C09042=1045.167,89.318,-85.987,170.316,36.397,156.850
C09043=1045.173,89.567,-86.006,170.318,36.398,156.851
C09044=1045.179,89.816,-86.025,170.319,36.400,156.851
C09045=1045.185,90.066,-86.044,170.321,36.401,156.851
C09046=1045.192,90.315,-86.063,170.324,36.403,156.851
C09047=1045.198,90.564,-86.081,170.325,36.404,156.852
C09048=1045.204,90.813,-86.101,170.327,36.406,156.852
C09049=1045.210,91.062,-86.119,170.329,36.407,156.852
C09050=1045.216,91.312,-86.138,170.330,36.408,156.853
C09051=1045.223,91.560,-86.158,170.332,36.410,156.853
C09052=1045.228,91.810,-86.177,170.334,36.411,156.853
C09053=1045.234,92.059,-86.196,170.336,36.413,156.853
C09054=1045.240,92.308,-86.215,170.338,36.415,156.854
C09055=1045.247,92.558,-86.235,170.340,36.416,156.854
C09056=1045.253,92.807,-86.254,170.341,36.417,156.854
C09057=1045.260,93.093,-86.275,170.343,36.419,156.855
C09058=1045.267,93.379,-86.297,170.346,36.421,156.855
C09059=1045.274,93.665,-86.319,170.348,36.422,156.855
C09060=1045.281,93.951,-86.341,170.350,36.424,156.855
C09061=1045.288,94.200,-86.361,170.352,36.425,156.856
C09062=1045.293,94.449,-86.380,170.353,36.426,156.856
C09063=1045.300,94.698,-86.399,170.355,36.428,156.856
C09064=1045.305,94.948,-86.418,170.357,36.430,156.857
C09065=1045.312,95.196,-86.437,170.359,36.431,156.857
C09066=1045.318,95.446,-86.456,170.361,36.433,156.857
C09067=1045.324,95.695,-86.475,170.363,36.434,156.857
C09068=1045.331,95.944,-86.495,170.365,36.435,156.858
C09069=1045.337,96.193,-86.514,170.366,36.437,156.858
C09070=1045.343,96.443,-86.533,170.368,36.438,156.858
C09071=1045.349,96.692,-86.553,170.371,36.440,156.858
C09072=1045.355,96.941,-86.572,170.372,36.441,156.859
C09073=1045.361,97.190,-86.591,170.374,36.443,156.859
C09074=1045.368,97.439,-86.611,170.376,36.444,156.859
C09075=1045.373,97.688,-86.630,170.377,36.445,156.860
C09076=1045.381,97.938,-86.649,170.379,36.447,156.860
C09077=1045.386,98.153,-86.666,170.381,36.448,156.860
C09078=1045.391,98.367,-86.683,170.383,36.450,156.860
C09079=1045.396,98.582,-86.699,170.384,36.451,156.861
C09080=1045.401,98.797,-86.715,170.386,36.452,156.861
C09081=1045.407,99.011,-86.732,170.387,36.453,156.861
C09082=1045.412,99.227,-86.749,170.389,36.454,156.861
C09083=1045.418,99.441,-86.765,170.390,36.455,156.861
C09084=1045.423,99.655,-86.782,170.392,36.456,156.862
C09085=1045.429,99.905,-86.802,170.394,36.458,156.862
C09086=1045.436,100.153,-86.821,170.396,36.460,156.862
C09087=1045.442,100.403,-86.841,170.398,36.461,156.863
C09088=1045.448,100.653,-86.860,170.399,36.462,156.863
C09089=1045.454,100.901,-86.879,170.401,36.464,156.863
C09090=1045.460,101.150,-86.899,170.403,36.465,156.863
C09091=1045.466,101.400,-86.918,170.405,36.467,156.864
C09092=1045.472,101.648,-86.938,170.407,36.468,156.864
C09093=1045.478,101.899,-86.958,170.409,36.470,156.864
C09094=1045.485,102.147,-86.977,170.411,36.471,156.865
C09095=1045.491,102.397,-86.997,170.412,36.473,156.865
C09096=1045.497,102.645,-87.016,170.415,36.474,156.865
C09097=1045.503,102.895,-87.036,170.417,36.476,156.865
C09098=1045.509,103.144,-87.056,170.418,36.477,156.866
C09099=1045.515,103.394,-87.075,170.420,36.479,156.866
C09100=1045.522,103.642,-87.095,170.422,36.480,156.866
C09101=1045.528,103.891,-87.115,170.423,36.482,156.867
C09102=1045.533,104.140,-87.134,170.426,36.483,156.867
C09103=1045.539,104.389,-87.154,170.428,36.484,156.867
C09104=1045.546,104.639,-87.173,170.429,36.486,156.867
C09105=1045.552,104.888,-87.193,170.431,36.488,156.868
C09106=1045.558,105.137,-87.213,170.433,36.489,156.868
C09107=1045.564,105.386,-87.232,170.434,36.491,156.868
C09108=1045.571,105.636,-87.252,170.437,36.492,156.868
C09109=1045.577,105.885,-87.272,170.439,36.494,156.869
C09110=1045.582,106.134,-87.292,170.441,36.495,156.869
C09111=1045.588,106.383,-87.311,170.442,36.496,156.869
C09112=1045.596,106.632,-87.331,170.444,36.498,156.870
C09113=1045.601,106.881,-87.350,170.446,36.499,156.870
C09114=1045.607,107.130,-87.370,170.448,36.501,156.870
C09115=1045.613,107.379,-87.390,170.450,36.503,156.871
C09116=1045.620,107.629,-87.410,170.452,36.504,156.871
C09117=1045.626,107.878,-87.430,170.453,36.506,156.871
C09118=1045.632,108.126,-87.449,170.455,36.507,156.871
C09119=1045.639,108.376,-87.470,170.457,36.508,156.872
C09120=1045.645,108.625,-87.489,170.460,36.510,156.872
C09121=1045.654,108.980,-87.517,170.462,36.512,156.872
C09122=1045.662,109.335,-87.546,170.464,36.514,156.873
C09123=1045.671,109.689,-87.574,170.467,36.516,156.873
C09124=1045.680,110.044,-87.602,170.469,36.518,156.874
C09125=1045.686,110.294,-87.622,170.472,36.519,156.874
C09126=1045.692,110.542,-87.642,170.474,36.521,156.874
C09127=1045.698,110.791,-87.662,170.476,36.522,156.874
C09128=1045.705,111.041,-87.682,170.477,36.524,156.875
C09129=1045.711,111.290,-87.702,170.479,36.526,156.875
C09130=1045.716,111.539,-87.721,170.482,36.527,156.875
C09131=1045.723,111.789,-87.741,170.483,36.529,156.876
C09132=1045.729,112.037,-87.761,170.485,36.530,156.876
C09133=1045.735,112.286,-87.781,170.487,36.532,156.876
C09134=1045.742,112.536,-87.802,170.488,36.533,156.876
C09135=1045.748,112.785,-87.822,170.490,36.534,156.877
C09136=1045.754,113.033,-87.842,170.493,36.536,156.877
C09137=1045.760,113.283,-87.862,170.495,36.537,156.877
C09138=1045.766,113.532,-87.882,170.496,36.539,156.878
C09139=1045.772,113.780,-87.902,170.498,36.540,156.878
C09140=1045.778,114.031,-87.921,170.500,36.542,156.878
C09141=1045.784,114.280,-87.942,170.501,36.544,156.878
C09142=1045.790,114.529,-87.962,170.504,36.545,156.879
C09143=1045.796,114.778,-87.982,170.506,36.547,156.879
C09144=1045.803,115.026,-88.003,170.508,36.548,156.879
C09145=1045.808,115.275,-88.024,170.509,36.550,156.880
C09146=1045.814,115.525,-88.044,170.511,36.552,156.880
C09147=1045.820,115.774,-88.064,170.514,36.553,156.880
C09148=1045.826,116.023,-88.084,170.515,36.555,156.881
C09149=1045.832,116.272,-88.105,170.517,36.556,156.881
C09150=1045.838,116.521,-88.125,170.519,36.558,156.881
C09151=1045.844,116.770,-88.145,170.520,36.559,156.881
C09152=1045.850,117.020,-88.166,170.522,36.561,156.882
C09153=1045.856,117.269,-88.185,170.525,36.562,156.882
C09154=1045.862,117.517,-88.205,170.527,36.564,156.882
C09155=1045.868,117.767,-88.226,170.528,36.566,156.883
C09156=1045.874,118.016,-88.246,170.530,36.567,156.883
C09157=1045.880,118.265,-88.266,170.532,36.569,156.883
C09158=1045.887,118.514,-88.287,170.535,36.570,156.884
C09159=1045.892,118.763,-88.308,170.536,36.572,156.884
C09160=1045.899,119.012,-88.328,170.538,36.573,156.884
C09161=1045.905,119.261,-88.348,170.540,36.575,156.885
C09162=1045.910,119.510,-88.369,170.541,36.576,156.885
C09163=1045.917,119.760,-88.389,170.544,36.578,156.885
C09164=1045.923,120.009,-88.409,170.546,36.579,156.885
C09165=1045.929,120.258,-88.430,170.548,36.581,156.886
C09166=1045.935,120.507,-88.451,170.549,36.583,156.886
C09167=1045.941,120.756,-88.471,170.551,36.584,156.886
C09168=1045.947,121.005,-88.491,170.553,36.586,156.887
C09169=1045.953,121.254,-88.511,170.556,36.588,156.887
C09170=1045.959,121.503,-88.532,170.557,36.589,156.887
C09171=1045.965,121.752,-88.552,170.559,36.591,156.888
C09172=1045.971,122.002,-88.573,170.561,36.592,156.888
C09173=1045.977,122.251,-88.593,170.562,36.594,156.888
C09174=1045.984,122.499,-88.614,170.564,36.595,156.888
C09175=1045.989,122.749,-88.635,170.567,36.597,156.889
C09176=1045.996,122.998,-88.655,170.569,36.598,156.889
C09177=1046.002,123.247,-88.675,170.570,36.600,156.889
C09178=1046.008,123.496,-88.697,170.572,36.601,156.890
C09179=1046.014,123.745,-88.717,170.574,36.603,156.890
C09180=1046.021,123.994,-88.737,170.577,36.604,156.890
C09181=1046.026,124.243,-88.758,170.579,36.606,156.891
C09182=1046.033,124.492,-88.779,170.580,36.607,156.891
C09183=1046.039,124.741,-88.799,170.582,36.609,156.891
C09184=1046.045,124.990,-88.820,170.584,36.610,156.891
C09185=1046.052,125.276,-88.843,170.587,36.612,156.892
C09186=1046.059,125.562,-88.867,170.589,36.614,156.892
C09187=1046.066,125.848,-88.891,170.591,36.616,156.893
C09188=1046.073,126.133,-88.915,170.593,36.617,156.893
C09189=1046.079,126.382,-88.935,170.595,36.619,156.893
C09190=1046.085,126.632,-88.955,170.597,36.620,156.893
C09191=1046.092,126.881,-88.976,170.599,36.622,156.894
C09192=1046.098,127.130,-88.996,170.601,36.623,156.894
C09193=1046.104,127.379,-89.018,170.603,36.625,156.894
C09194=1046.110,127.628,-89.038,170.605,36.626,156.895
C09195=1046.117,127.877,-89.058,170.606,36.628,156.895
C09196=1046.122,128.126,-89.080,170.609,36.630,156.895
C09197=1046.129,128.375,-89.100,170.611,36.631,156.896
C09198=1046.135,128.624,-89.122,170.613,36.633,156.896
C09199=1046.141,128.873,-89.142,170.615,36.634,156.896
C09200=1046.148,129.122,-89.163,170.616,36.636,156.896
C09201=1046.153,129.371,-89.183,170.619,36.637,156.897
C09202=1046.160,129.620,-89.204,170.621,36.639,156.897
C09203=1046.167,129.870,-89.225,170.623,36.640,156.897
C09204=1046.172,130.118,-89.246,170.624,36.642,156.898
C09205=1046.179,130.368,-89.266,170.626,36.643,156.898
C09206=1046.185,130.616,-89.287,170.629,36.645,156.898
C09207=1046.191,130.866,-89.308,170.631,36.646,156.898
C09208=1046.198,131.115,-89.329,170.633,36.648,156.899
C09209=1046.203,131.364,-89.349,170.634,36.649,156.899
C09210=1046.210,131.613,-89.370,170.636,36.651,156.899
C09211=1046.216,131.862,-89.391,170.638,36.652,156.900
C09212=1046.222,132.111,-89.413,170.641,36.654,156.900
C09213=1046.229,132.360,-89.434,170.643,36.656,156.900
C09214=1046.234,132.609,-89.454,170.644,36.657,156.901
C09215=1046.240,132.858,-89.476,170.646,36.659,156.901
C09216=1046.247,133.107,-89.497,170.648,36.660,156.901
C09217=1046.252,133.356,-89.517,170.651,36.662,156.902
C09218=1046.258,133.605,-89.539,170.653,36.664,156.902
C09219=1046.265,133.854,-89.560,170.654,36.665,156.902
C09220=1046.270,134.103,-89.581,170.656,36.667,156.903
C09221=1046.277,134.353,-89.602,170.658,36.668,156.903
C09222=1046.283,134.601,-89.623,170.661,36.670,156.903
C09223=1046.289,134.851,-89.644,170.663,36.672,156.904
C09224=1046.295,135.100,-89.665,170.664,36.673,156.904
C09225=1046.300,135.348,-89.687,170.666,36.675,156.904
C09226=1046.307,135.597,-89.708,170.668,36.676,156.904
C09227=1046.313,135.847,-89.729,170.671,36.678,156.905
C09228=1046.319,136.096,-89.750,170.673,36.680,156.905
C09229=1046.326,136.344,-89.771,170.674,36.681,156.905
C09230=1046.332,136.594,-89.793,170.676,36.683,156.906
C09231=1046.337,136.843,-89.813,170.678,36.684,156.906
C09232=1046.344,137.092,-89.834,170.681,36.686,156.906
C09233=1046.350,137.341,-89.856,170.683,36.688,156.907
C09234=1046.356,137.589,-89.877,170.684,36.689,156.907
C09235=1046.362,137.839,-89.899,170.686,36.691,156.907
C09236=1046.369,138.088,-89.920,170.688,36.693,156.908
C09237=1046.374,138.337,-89.940,170.691,36.694,156.908
C09238=1046.380,138.586,-89.962,170.693,36.696,156.908
C09239=1046.386,138.835,-89.984,170.695,36.697,156.909
C09240=1046.393,139.084,-90.005,170.696,36.699,156.909
C09241=1046.399,139.332,-90.026,170.698,36.701,156.909
C09242=1046.405,139.582,-90.048,170.701,36.702,156.910
C09243=1046.411,139.831,-90.069,170.703,36.704,156.910
C09244=1046.417,140.079,-90.090,170.705,36.706,156.910
C09245=1046.423,140.329,-90.111,170.706,36.707,156.911
C09246=1046.429,140.578,-90.133,170.708,36.709,156.911
C09247=1046.435,140.828,-90.155,170.711,36.711,156.911
C09248=1046.440,141.076,-90.176,170.713,36.712,156.912
C09249=1046.448,141.362,-90.201,170.715,36.714,156.912
C09250=1046.455,141.647,-90.225,170.717,36.716,156.912
C09251=1046.462,141.933,-90.250,170.720,36.718,156.913
C09252=1046.469,142.218,-90.275,170.722,36.720,156.913
C09253=1046.475,142.467,-90.296,170.724,36.721,156.913
C09254=1046.481,142.716,-90.318,170.726,36.723,156.914
C09255=1046.487,142.965,-90.339,170.728,36.725,156.914
C09256=1046.493,143.214,-90.361,170.731,36.727,156.914
C09257=1046.499,143.463,-90.382,170.733,36.728,156.915
C09258=1046.506,143.712,-90.404,170.734,36.730,156.915
C09259=1046.511,143.961,-90.425,170.736,36.732,156.915
C09260=1046.517,144.210,-90.447,170.738,36.733,156.916
C09261=1046.523,144.459,-90.469,170.741,36.735,156.916
C09262=1046.530,144.708,-90.490,170.743,36.737,156.916
C09263=1046.536,144.958,-90.512,170.745,36.738,156.917
C09264=1046.541,145.206,-90.533,170.746,36.740,156.917
C09265=1046.547,145.455,-90.555,170.748,36.741,156.917
C09266=1046.554,145.704,-90.577,170.751,36.743,156.918
C09267=1046.560,145.953,-90.599,170.753,36.745,156.918
C09268=1046.566,146.202,-90.620,170.755,36.746,156.918
C09269=1046.572,146.451,-90.642,170.757,36.748,156.919
C09270=1046.578,146.700,-90.663,170.759,36.749,156.919
C09271=1046.585,146.949,-90.684,170.762,36.751,156.919
C09272=1046.591,147.198,-90.706,170.763,36.753,156.920
C09273=1046.597,147.447,-90.729,170.765,36.754,156.920
C09274=1046.603,147.696,-90.751,170.767,36.756,156.920
C09275=1046.609,147.945,-90.772,170.770,36.758,156.921
C09276=1046.615,148.194,-90.793,170.772,36.760,156.921
C09277=1046.621,148.443,-90.816,170.774,36.761,156.921
C09278=1046.627,148.692,-90.837,170.776,36.763,156.922
C09279=1046.633,148.941,-90.859,170.777,36.765,156.922
C09280=1046.640,149.190,-90.881,170.780,36.767,156.922
C09281=1046.645,149.439,-90.904,170.782,36.768,156.923
C09282=1046.651,149.688,-90.925,170.784,36.770,156.923
C09283=1046.657,149.937,-90.947,170.786,36.771,156.923
C09284=1046.664,150.185,-90.969,170.788,36.773,156.924
C09285=1046.670,150.435,-90.991,170.791,36.775,156.924
C09286=1046.676,150.684,-91.012,170.793,36.776,156.924
C09287=1046.682,150.933,-91.035,170.795,36.778,156.925
C09288=1046.688,151.182,-91.057,170.796,36.780,156.925
C09289=1046.693,151.430,-91.078,170.799,36.782,156.925
C09290=1046.700,151.679,-91.100,170.801,36.784,156.926
C09291=1046.705,151.929,-91.123,170.803,36.785,156.926
C09292=1046.711,152.178,-91.144,170.805,36.787,156.926
C09293=1046.718,152.426,-91.167,170.807,36.789,156.927
C09294=1046.724,152.676,-91.188,170.810,36.790,156.927
C09295=1046.731,152.924,-91.211,170.812,36.792,156.928
C09296=1046.736,153.174,-91.233,170.814,36.793,156.928
C09297=1046.742,153.422,-91.255,170.815,36.795,156.928
C09298=1046.749,153.671,-91.277,170.818,36.797,156.929
C09299=1046.754,153.920,-91.298,170.820,36.799,156.929
C09300=1046.760,154.169,-91.321,170.822,36.801,156.929
C09301=1046.766,154.418,-91.343,170.824,36.802,156.930
C09302=1046.772,154.667,-91.365,170.826,36.804,156.930
C09303=1046.779,154.916,-91.387,170.829,36.806,156.930
C09304=1046.784,155.165,-91.410,170.831,36.808,156.931
C09305=1046.791,155.414,-91.431,170.833,36.809,156.931
C09306=1046.796,155.663,-91.454,170.835,36.811,156.931
C09307=1046.803,155.911,-91.477,170.838,36.813,156.932
C09308=1046.809,156.161,-91.498,170.839,36.814,156.932
C09309=1046.815,156.410,-91.521,170.841,36.816,156.932
C09310=1046.821,156.659,-91.543,170.843,36.818,156.933
C09311=1046.827,156.907,-91.565,170.845,36.820,156.933
C09312=1046.833,157.157,-91.587,170.848,36.822,156.933
C09313=1046.840,157.441,-91.613,170.850,36.823,156.934
C09314=1046.847,157.727,-91.638,170.853,36.825,156.934
C09315=1046.854,158.012,-91.664,170.855,36.828,156.935
C09316=1046.861,158.297,-91.689,170.858,36.829,156.935
C09317=1046.867,158.546,-91.712,170.860,36.831,156.935
C09318=1046.873,158.795,-91.734,170.862,36.833,156.936
C09319=1046.879,159.044,-91.756,170.864,36.835,156.936
C09320=1046.885,159.293,-91.779,170.867,36.837,156.937
C09321=1046.891,159.542,-91.801,170.869,36.838,156.937
C09322=1046.897,159.791,-91.824,170.871,36.840,156.937
C09323=1046.903,160.040,-91.846,170.873,36.842,156.938
C09324=1046.910,160.288,-91.869,170.876,36.843,156.938
C09325=1046.915,160.538,-91.891,170.878,36.845,156.938
C09326=1046.921,160.787,-91.914,170.879,36.847,156.939
C09327=1046.927,161.035,-91.936,170.881,36.849,156.939
C09328=1046.933,161.284,-91.959,170.883,36.851,156.939
C09329=1046.939,161.534,-91.981,170.886,36.853,156.940
C09330=1046.944,161.782,-92.004,170.888,36.854,156.940
C09331=1046.951,162.031,-92.027,170.890,36.856,156.941
C09332=1046.956,162.280,-92.049,170.893,36.859,156.941
C09333=1046.962,162.529,-92.072,170.895,36.861,156.941
C09334=1046.968,162.778,-92.095,170.897,36.862,156.942
C09335=1046.974,163.027,-92.118,170.899,36.864,156.942
C09336=1046.980,163.275,-92.141,170.901,36.866,156.942
C09337=1046.986,163.525,-92.163,170.904,36.868,156.943
C09338=1046.991,163.774,-92.186,170.906,36.870,156.943
C09339=1046.997,164.023,-92.209,170.908,36.872,156.944
C09340=1047.003,164.271,-92.232,170.910,36.873,156.944
C09341=1047.009,164.520,-92.254,170.913,36.875,156.944
C09342=1047.015,164.769,-92.277,170.914,36.877,156.945
C09343=1047.021,165.018,-92.300,170.916,36.879,156.945
C09344=1047.026,165.267,-92.323,170.918,36.881,156.946
C09345=1047.032,165.516,-92.346,170.921,36.883,156.946
C09346=1047.039,165.764,-92.368,170.923,36.885,156.946
C09347=1047.045,166.014,-92.392,170.925,36.887,156.947
C09348=1047.051,166.263,-92.414,170.927,36.889,156.947
C09349=1047.056,166.512,-92.437,170.930,36.890,156.947
C09350=1047.062,166.761,-92.460,170.932,36.892,156.948
C09351=1047.069,167.009,-92.483,170.934,36.894,156.948
C09352=1047.074,167.258,-92.506,170.936,36.896,156.949
C09353=1047.080,167.507,-92.529,170.939,36.898,156.949
C09354=1047.086,167.756,-92.552,170.941,36.899,156.949
C09355=1047.092,168.005,-92.574,170.943,36.902,156.950
C09356=1047.098,168.253,-92.597,170.945,36.904,156.950
C09357=1047.105,168.502,-92.621,170.948,36.906,156.951
C09358=1047.110,168.751,-92.644,170.950,36.907,156.951
C09359=1047.116,169.000,-92.667,170.952,36.909,156.951
C09360=1047.122,169.249,-92.690,170.954,36.911,156.952
C09361=1047.128,169.498,-92.713,170.957,36.913,156.952
C09362=1047.134,169.746,-92.735,170.959,36.915,156.952
C09363=1047.140,169.995,-92.758,170.961,36.916,156.953
C09364=1047.146,170.244,-92.782,170.963,36.918,156.953
C09365=1047.152,170.493,-92.805,170.966,36.921,156.954
C09366=1047.158,170.742,-92.828,170.968,36.923,156.954
C09367=1047.164,170.991,-92.851,170.970,36.924,156.954
C09368=1047.170,171.240,-92.873,170.972,36.926,156.955
C09369=1047.176,171.489,-92.896,170.975,36.928,156.955
C09370=1047.182,171.737,-92.920,170.977,36.930,156.956
C09371=1047.188,171.986,-92.943,170.979,36.932,156.956
C09372=1047.194,172.235,-92.966,170.981,36.933,156.956
C09373=1047.200,172.484,-92.989,170.984,36.935,156.957
C09374=1047.206,172.733,-93.013,170.986,36.937,156.957
C09375=1047.213,172.982,-93.035,170.988,36.940,156.957
C09376=1047.218,173.231,-93.058,170.991,36.941,156.958
C09377=1047.225,173.515,-93.086,170.994,36.943,156.958
C09378=1047.232,173.800,-93.111,170.996,36.946,156.959
C09379=1047.239,174.085,-93.138,170.999,36.947,156.959
C09380=1047.246,174.370,-93.165,171.002,36.950,156.960
C09381=1047.253,174.619,-93.188,171.004,36.952,156.960
C09382=1047.258,174.868,-93.211,171.006,36.953,156.960
C09383=1047.264,175.116,-93.234,171.008,36.955,156.961
C09384=1047.271,175.366,-93.258,171.011,36.957,156.961
C09385=1047.276,175.614,-93.281,171.013,36.959,156.962
C09386=1047.283,175.863,-93.304,171.015,36.961,156.962
C09387=1047.288,176.112,-93.327,171.018,36.963,156.962
C09388=1047.295,176.361,-93.351,171.020,36.965,156.963
C09389=1047.301,176.610,-93.374,171.023,36.967,156.963
C09390=1047.307,176.858,-93.396,171.025,36.969,156.963
C09391=1047.314,177.107,-93.421,171.028,36.970,156.964
C09392=1047.319,177.356,-93.443,171.030,36.972,156.964
C09393=1047.325,177.604,-93.467,171.032,36.975,156.965
C09394=1047.332,177.854,-93.490,171.034,36.976,156.965
C09395=1047.338,178.102,-93.514,171.037,36.978,156.965
C09396=1047.344,178.352,-93.537,171.039,36.980,156.966
C09397=1047.350,178.600,-93.561,171.041,36.982,156.966
C09398=1047.356,178.849,-93.584,171.043,36.984,156.967
C09399=1047.363,179.098,-93.608,171.046,36.985,156.967
C09400=1047.368,179.347,-93.631,171.049,36.988,156.967
C09401=1047.375,179.595,-93.654,171.051,36.990,156.968
C09402=1047.381,179.844,-93.677,171.053,36.991,156.968
C09403=1047.387,180.093,-93.701,171.056,36.993,156.969
C09404=1047.394,180.342,-93.724,171.058,36.995,156.969
C09405=1047.400,180.590,-93.748,171.060,36.997,156.969
C09406=1047.406,180.839,-93.771,171.062,36.999,156.970
C09407=1047.412,181.088,-93.795,171.065,37.001,156.970
C09408=1047.418,181.337,-93.819,171.068,37.003,156.971
C09409=1047.425,181.586,-93.842,171.070,37.005,156.971
C09410=1047.431,181.835,-93.866,171.073,37.007,156.971
C09411=1047.437,182.084,-93.889,171.075,37.008,156.972
C09412=1047.443,182.332,-93.913,171.077,37.011,156.972
C09413=1047.450,182.581,-93.937,171.079,37.013,156.973
C09414=1047.455,182.830,-93.960,171.082,37.014,156.973
C09415=1047.462,183.079,-93.984,171.085,37.016,156.973
C09416=1047.469,183.327,-94.007,171.087,37.018,156.974
C09417=1047.475,183.577,-94.030,171.089,37.020,156.974
C09418=1047.481,183.825,-94.054,171.092,37.022,156.975
C09419=1047.486,184.074,-94.078,171.094,37.024,156.975
C09420=1047.493,184.323,-94.102,171.096,37.026,156.975
C09421=1047.498,184.572,-94.125,171.099,37.028,156.976
C09422=1047.505,184.821,-94.149,171.102,37.030,156.976
C09423=1047.510,185.069,-94.174,171.104,37.032,156.977
C09424=1047.516,185.318,-94.197,171.106,37.034,156.977
C09425=1047.523,185.567,-94.221,171.109,37.037,156.978
C09426=1047.528,185.815,-94.246,171.111,37.038,156.978
C09427=1047.535,186.064,-94.270,171.113,37.041,156.978
C09428=1047.540,186.313,-94.293,171.116,37.043,156.979
C09429=1047.546,186.562,-94.317,171.118,37.045,156.979
C09430=1047.552,186.811,-94.342,171.121,37.047,156.980
C09431=1047.558,187.059,-94.365,171.123,37.049,156.980
C09432=1047.563,187.309,-94.390,171.126,37.051,156.981
C09433=1047.570,187.557,-94.413,171.128,37.054,156.981
C09434=1047.575,187.806,-94.438,171.130,37.055,156.982
C09435=1047.581,188.054,-94.462,171.133,37.058,156.982
C09436=1047.587,188.304,-94.486,171.135,37.060,156.982
C09437=1047.593,188.552,-94.510,171.138,37.062,156.983
C09438=1047.599,188.801,-94.534,171.141,37.064,156.983
C09439=1047.605,189.050,-94.558,171.143,37.066,156.984
C09440=1047.611,189.298,-94.583,171.145,37.068,156.984
C09441=1047.618,189.582,-94.611,171.148,37.070,156.985
C09442=1047.625,189.867,-94.638,171.151,37.073,156.985
C09443=1047.631,190.151,-94.665,171.154,37.075,156.986
C09444=1047.638,190.436,-94.694,171.156,37.078,156.986
C09445=1047.645,190.685,-94.718,171.159,37.080,156.987
C09446=1047.650,190.933,-94.742,171.161,37.082,156.987
C09447=1047.657,191.182,-94.766,171.164,37.084,156.988
C09448=1047.662,191.431,-94.790,171.167,37.086,156.988
C09449=1047.669,191.680,-94.814,171.169,37.088,156.988
C09450=1047.674,191.929,-94.839,171.171,37.090,156.989
C09451=1047.681,192.177,-94.863,171.174,37.093,156.989
C09452=1047.687,192.426,-94.888,171.177,37.094,156.990
C09453=1047.693,192.675,-94.912,171.179,37.097,156.990
C09454=1047.699,192.924,-94.936,171.182,37.099,156.991
C09455=1047.705,193.172,-94.960,171.184,37.101,156.991
C09456=1047.711,193.421,-94.985,171.186,37.103,156.992
C09457=1047.717,193.669,-95.009,171.189,37.105,156.992
C09458=1047.723,193.918,-95.033,171.192,37.108,156.992
C09459=1047.730,194.167,-95.057,171.194,37.109,156.993
C09460=1047.735,194.416,-95.082,171.196,37.112,156.993
C09461=1047.741,194.665,-95.107,171.200,37.114,156.994
C09462=1047.748,194.914,-95.131,171.202,37.116,156.994
C09463=1047.753,195.162,-95.155,171.204,37.118,156.995
C09464=1047.760,195.411,-95.179,171.207,37.120,156.995
C09465=1047.765,195.659,-95.204,171.209,37.123,156.996
C09466=1047.772,195.908,-95.228,171.212,37.124,156.996
C09467=1047.778,196.157,-95.253,171.215,37.127,156.996
C09468=1047.785,196.406,-95.278,171.217,37.129,156.997
C09469=1047.790,196.654,-95.302,171.219,37.131,156.997
C09470=1047.796,196.904,-95.327,171.222,37.133,156.998
C09471=1047.803,197.152,-95.351,171.225,37.135,156.998
C09472=1047.808,197.401,-95.376,171.227,37.138,156.999
C09473=1047.815,197.649,-95.400,171.230,37.140,156.999
C09474=1047.821,197.898,-95.425,171.233,37.142,157.000
C09475=1047.827,198.146,-95.449,171.235,37.144,157.000
C09476=1047.833,198.395,-95.474,171.237,37.146,157.001
C09477=1047.839,198.644,-95.499,171.241,37.148,157.001
C09478=1047.846,198.893,-95.523,171.243,37.151,157.002
C09479=1047.851,199.141,-95.548,171.245,37.153,157.002
C09480=1047.858,199.390,-95.572,171.249,37.155,157.002
C09481=1047.864,199.639,-95.597,171.251,37.157,157.003
C09482=1047.870,199.888,-95.622,171.253,37.159,157.003
C09483=1047.876,200.136,-95.646,171.256,37.162,157.004
C09484=1047.882,200.385,-95.671,171.259,37.163,157.004
C09485=1047.889,200.634,-95.695,171.261,37.166,157.005
C09486=1047.895,200.883,-95.720,171.264,37.168,157.005
C09487=1047.901,201.132,-95.745,171.267,37.170,157.006
C09488=1047.908,201.379,-95.770,171.269,37.172,157.006
C09489=1047.914,201.628,-95.794,171.272,37.175,157.007
C09490=1047.920,201.877,-95.820,171.275,37.177,157.007
C09491=1047.926,202.126,-95.844,171.277,37.179,157.008
C09492=1047.931,202.374,-95.869,171.279,37.181,157.008
C09493=1047.938,202.623,-95.895,171.282,37.184,157.009
C09494=1047.943,202.872,-95.919,171.285,37.186,157.009
C09495=1047.950,203.121,-95.945,171.288,37.188,157.010
C09496=1047.957,203.369,-95.969,171.290,37.191,157.010
C09497=1047.962,203.618,-95.994,171.293,37.193,157.010
C09498=1047.968,203.867,-96.019,171.296,37.195,157.011
C09499=1047.974,204.115,-96.044,171.298,37.197,157.011
C09500=1047.981,204.364,-96.070,171.301,37.200,157.012
C09501=1047.986,204.613,-96.094,171.304,37.202,157.012
C09502=1047.992,204.861,-96.119,171.306,37.205,157.013
C09503=1047.998,205.110,-96.144,171.309,37.207,157.013
C09504=1048.004,205.359,-96.170,171.312,37.209,157.014
C09505=1048.030,206.410,-96.276,171.553,37.308,157.036
C09506=1048.037,206.675,-96.304,171.556,37.311,157.037
C09507=1048.044,206.939,-96.331,171.558,37.314,157.038
C09508=1048.051,207.204,-96.359,171.560,37.317,157.038
C09509=1048.058,207.469,-96.387,171.562,37.321,157.039
C09510=1048.065,207.717,-96.413,171.565,37.324,157.040
C09511=1048.071,207.965,-96.439,171.566,37.327,157.040
C09512=1048.077,208.215,-96.466,171.569,37.330,157.041
C09513=1048.084,208.463,-96.492,171.570,37.333,157.042
C09514=1048.091,208.711,-96.518,171.573,37.336,157.042
C09515=1048.097,208.960,-96.544,171.574,37.339,157.043
C09516=1048.103,209.208,-96.571,171.576,37.342,157.044
C09517=1048.110,209.457,-96.597,171.579,37.345,157.044
C09518=1048.117,209.705,-96.623,171.580,37.348,157.045
C09519=1048.123,209.954,-96.650,171.583,37.352,157.046
C09520=1048.129,210.202,-96.676,171.584,37.355,157.046
C09521=1048.136,210.451,-96.703,171.587,37.358,157.047
C09522=1048.142,210.700,-96.729,171.588,37.361,157.048
C09523=1048.149,210.948,-96.755,171.591,37.364,157.048
C09524=1048.155,211.197,-96.782,171.593,37.367,157.049
C09525=1048.162,211.445,-96.808,171.595,37.370,157.050
C09526=1048.169,211.693,-96.834,171.597,37.373,157.050
C09527=1048.175,211.942,-96.861,171.599,37.376,157.051
C09528=1048.182,212.191,-96.887,171.601,37.379,157.052
C09529=1048.187,212.439,-96.914,171.604,37.382,157.052
C09530=1048.195,212.688,-96.941,171.605,37.386,157.053
C09531=1048.200,212.936,-96.967,171.608,37.389,157.054
C09532=1048.207,213.185,-96.994,171.609,37.392,157.054
C09533=1048.213,213.433,-97.020,171.612,37.395,157.055
C09534=1048.220,213.682,-97.047,171.614,37.398,157.055
C09535=1048.226,213.930,-97.073,171.616,37.401,157.056
C09536=1048.232,214.179,-97.100,171.618,37.404,157.057
C09537=1048.239,214.427,-97.126,171.619,37.407,157.058
C09538=1048.246,214.676,-97.154,171.622,37.410,157.058
C09539=1048.252,214.924,-97.180,171.624,37.413,157.059
C09540=1048.259,215.173,-97.207,171.626,37.416,157.059
C09541=1048.264,215.421,-97.234,171.628,37.420,157.060
C09542=1048.271,215.670,-97.260,171.631,37.423,157.061
C09543=1048.277,215.918,-97.287,171.632,37.426,157.061
C09544=1048.284,216.167,-97.313,171.635,37.429,157.062
C09545=1048.290,216.415,-97.341,171.637,37.432,157.063
C09546=1048.298,216.664,-97.367,171.639,37.435,157.063
C09547=1048.303,216.912,-97.394,171.641,37.438,157.064
C09548=1048.310,217.161,-97.421,171.643,37.441,157.065
C09549=1048.316,217.409,-97.447,171.645,37.444,157.065
C09550=1048.323,217.658,-97.475,171.648,37.447,157.066
C09551=1048.330,217.906,-97.501,171.649,37.450,157.067
C09552=1048.336,218.155,-97.528,171.652,37.453,157.067
C09553=1048.342,218.404,-97.555,171.654,37.456,157.068
C09554=1048.349,218.651,-97.581,171.656,37.459,157.069
C09555=1048.355,218.900,-97.608,171.658,37.462,157.069
C09556=1048.362,219.149,-97.635,171.661,37.465,157.070
C09557=1048.369,219.397,-97.662,171.663,37.468,157.071
C09558=1048.375,219.646,-97.689,171.665,37.471,157.071
C09559=1048.382,219.894,-97.716,171.667,37.474,157.072
C09560=1048.388,220.142,-97.743,171.670,37.477,157.073
C09561=1048.395,220.391,-97.769,171.671,37.480,157.073
C09562=1048.402,220.661,-97.799,171.673,37.483,157.074
C09563=1048.409,220.931,-97.828,171.676,37.487,157.075
C09564=1048.416,221.201,-97.857,171.679,37.490,157.075
C09565=1048.422,221.471,-97.887,171.681,37.493,157.076
C09566=1048.429,221.720,-97.914,171.683,37.496,157.077
C09567=1048.435,221.967,-97.941,171.685,37.499,157.077
C09568=1048.442,222.216,-97.968,171.688,37.503,157.078
C09569=1048.449,222.465,-97.996,171.689,37.506,157.079
C09570=1048.454,222.713,-98.022,171.692,37.509,157.079
C09571=1048.461,222.962,-98.050,171.694,37.512,157.080
C09572=1048.467,223.211,-98.077,171.697,37.515,157.081
C09573=1048.473,223.458,-98.104,171.698,37.518,157.081
C09574=1048.481,223.707,-98.131,171.700,37.521,157.082
C09575=1048.487,223.956,-98.159,171.703,37.524,157.083
C09576=1048.493,224.204,-98.185,171.705,37.527,157.083
C09577=1048.500,224.452,-98.213,171.707,37.530,157.084
C09578=1048.506,224.701,-98.241,171.709,37.533,157.085
C09579=1048.512,224.949,-98.267,171.712,37.536,157.085
C09580=1048.519,225.198,-98.295,171.713,37.539,157.086
C09581=1048.526,225.446,-98.322,171.716,37.542,157.087
C09582=1048.532,225.694,-98.349,171.718,37.545,157.087
C09583=1048.539,225.943,-98.377,171.721,37.548,157.088
C09584=1048.545,226.192,-98.404,171.722,37.552,157.089
C09585=1048.551,226.439,-98.431,171.725,37.554,157.089
C09586=1048.558,226.688,-98.459,171.727,37.557,157.090
C09587=1048.564,226.937,-98.486,171.730,37.560,157.091
C09588=1048.571,227.185,-98.513,171.732,37.563,157.091
C09589=1048.577,227.433,-98.541,171.734,37.566,157.092
C09590=1048.584,227.682,-98.567,171.736,37.569,157.093
C09591=1048.591,227.930,-98.595,171.739,37.572,157.093
C09592=1048.597,228.179,-98.623,171.741,37.575,157.094
C09593=1048.604,228.428,-98.650,171.743,37.578,157.095
C09594=1048.610,228.675,-98.677,171.745,37.581,157.095
C09595=1048.617,228.924,-98.705,171.748,37.584,157.096
C09596=1048.623,229.172,-98.733,171.750,37.587,157.097
C09597=1048.630,229.421,-98.760,171.753,37.590,157.097
C09598=1048.636,229.669,-98.787,171.754,37.593,157.098
C09599=1048.642,229.918,-98.815,171.757,37.596,157.099
C09600=1048.649,230.166,-98.842,171.759,37.599,157.099
C09601=1048.655,230.415,-98.871,171.762,37.602,157.100
C09602=1048.662,230.663,-98.898,171.764,37.605,157.101
C09603=1048.668,230.911,-98.926,171.766,37.608,157.101
C09604=1048.674,231.160,-98.953,171.768,37.611,157.102
C09605=1048.681,231.409,-98.981,171.771,37.614,157.102
C09606=1048.688,231.657,-99.008,171.773,37.618,157.103
C09607=1048.694,231.905,-99.036,171.776,37.621,157.104
C09608=1048.700,232.153,-99.063,171.777,37.624,157.105
C09609=1048.706,232.402,-99.092,171.780,37.627,157.105
C09610=1048.713,232.650,-99.119,171.782,37.629,157.106
C09611=1048.720,232.899,-99.147,171.785,37.632,157.107
C09612=1048.726,233.147,-99.175,171.787,37.635,157.107
C09613=1048.732,233.395,-99.203,171.790,37.638,157.108
C09614=1048.738,233.644,-99.231,171.791,37.641,157.108
C09615=1048.745,233.892,-99.258,171.794,37.645,157.109
C09616=1048.752,234.141,-99.286,171.796,37.648,157.110
C09617=1048.758,234.389,-99.314,171.799,37.651,157.111
C09618=1048.764,234.651,-99.344,171.801,37.654,157.111
C09619=1048.772,234.914,-99.373,171.804,37.657,157.112
C09620=1048.778,235.176,-99.403,171.806,37.660,157.113
C09621=1048.785,235.438,-99.432,171.809,37.663,157.113
C09622=1048.791,235.687,-99.459,171.811,37.667,157.114
C09623=1048.797,235.936,-99.488,171.814,37.670,157.115
C09624=1048.804,236.183,-99.516,171.815,37.673,157.115
C09625=1048.811,236.432,-99.544,171.818,37.675,157.116
C09626=1048.818,236.680,-99.572,171.820,37.678,157.117
C09627=1048.824,236.929,-99.600,171.823,37.681,157.117
C09628=1048.830,237.178,-99.628,171.825,37.684,157.118
C09629=1048.837,237.426,-99.655,171.828,37.687,157.119
C09630=1048.843,237.673,-99.684,171.830,37.690,157.119
C09631=1048.849,237.922,-99.712,171.833,37.693,157.120
C09632=1048.856,238.170,-99.740,171.834,37.696,157.121
C09633=1048.862,238.419,-99.768,171.837,37.700,157.121
C09634=1048.869,238.667,-99.796,171.840,37.702,157.122
C09635=1048.876,238.915,-99.824,171.842,37.705,157.123
C09636=1048.882,239.164,-99.852,171.845,37.708,157.123
C09637=1048.888,239.413,-99.880,171.847,37.711,157.124
C09638=1048.895,239.660,-99.909,171.850,37.714,157.125
C09639=1048.901,239.909,-99.937,171.852,37.717,157.125
C09640=1048.908,240.158,-99.965,171.855,37.720,157.126
C09641=1048.915,240.406,-99.992,171.857,37.723,157.127
C09642=1048.921,240.654,-100.021,171.860,37.726,157.127
C09643=1048.928,240.903,-100.049,171.862,37.729,157.128
C09644=1048.934,241.151,-100.078,171.864,37.732,157.129
C09645=1048.940,241.399,-100.106,171.866,37.735,157.129
C09646=1048.947,241.648,-100.134,171.869,37.738,157.130
C09647=1048.953,241.896,-100.163,171.871,37.741,157.131
C09648=1048.959,242.144,-100.191,171.874,37.744,157.131
C09649=1048.966,242.392,-100.219,171.876,37.747,157.132
C09650=1048.972,242.641,-100.248,171.879,37.750,157.133
C09651=1048.979,242.889,-100.276,171.881,37.753,157.133
C09652=1048.985,243.138,-100.305,171.884,37.756,157.134
C09653=1048.991,243.386,-100.334,171.886,37.759,157.135
C09654=1048.998,243.634,-100.361,171.889,37.762,157.135
C09655=1049.004,243.882,-100.390,171.891,37.765,157.136
C09656=1049.011,244.131,-100.418,171.894,37.768,157.137
C09657=1049.017,244.379,-100.447,171.896,37.771,157.137
C09658=1049.023,244.628,-100.475,171.899,37.774,157.138
C09659=1049.030,244.875,-100.504,171.901,37.777,157.139
C09660=1049.036,245.124,-100.533,171.904,37.780,157.139
C09661=1049.043,245.372,-100.561,171.906,37.783,157.140
C09662=1049.049,245.620,-100.590,171.909,37.786,157.141
C09663=1049.055,245.869,-100.618,171.911,37.789,157.141
C09664=1049.062,246.117,-100.647,171.914,37.792,157.142
C09665=1049.069,246.365,-100.676,171.916,37.795,157.143
C09666=1049.075,246.614,-100.704,171.918,37.799,157.143
C09667=1049.081,246.862,-100.733,171.921,37.802,157.144
C09668=1049.087,247.110,-100.762,171.923,37.804,157.145
C09669=1049.093,247.358,-100.791,171.926,37.807,157.145
C09670=1049.099,247.607,-100.819,171.928,37.811,157.146
C09671=1049.105,247.855,-100.848,171.931,37.814,157.147
C09672=1049.112,248.103,-100.877,171.933,37.817,157.148
C09673=1049.119,248.352,-100.906,171.936,37.820,157.148
C09674=1049.125,248.608,-100.936,171.938,37.823,157.149
C09675=1049.132,248.865,-100.965,171.941,37.826,157.150
C09676=1049.138,249.121,-100.996,171.944,37.829,157.150
C09677=1049.145,249.378,-101.025,171.947,37.833,157.151
C09678=1049.151,249.626,-101.055,171.950,37.835,157.152
C09679=1049.158,249.875,-101.084,171.952,37.838,157.152
C09680=1049.164,250.123,-101.113,171.955,37.841,157.153
C09681=1049.171,250.370,-101.141,171.957,37.844,157.154
C09682=1049.177,250.619,-101.170,171.960,37.848,157.155
C09683=1049.183,250.867,-101.198,171.962,37.851,157.155
C09684=1049.189,251.115,-101.227,171.965,37.854,157.156
C09685=1049.196,251.364,-101.257,171.967,37.856,157.157
C09686=1049.202,251.612,-101.286,171.970,37.859,157.157
C09687=1049.209,251.861,-101.315,171.972,37.863,157.158
C09688=1049.215,252.109,-101.344,171.975,37.866,157.159
C09689=1049.221,252.357,-101.373,171.977,37.869,157.159
C09690=1049.228,252.605,-101.401,171.980,37.872,157.160
C09691=1049.235,252.853,-101.431,171.982,37.875,157.161
C09692=1049.241,253.102,-101.460,171.985,37.877,157.161
C09693=1049.248,253.350,-101.489,171.988,37.881,157.162
C09694=1049.254,253.598,-101.518,171.990,37.884,157.163
C09695=1049.260,253.846,-101.547,171.993,37.887,157.163
C09696=1049.267,254.095,-101.576,171.996,37.890,157.164
C09697=1049.273,254.343,-101.605,171.999,37.893,157.165
C09698=1049.279,254.591,-101.635,172.001,37.895,157.165
C09699=1049.286,254.839,-101.664,172.004,37.899,157.166
C09700=1049.293,255.087,-101.694,172.006,37.902,157.167
C09701=1049.299,255.336,-101.723,172.009,37.905,157.167
C09702=1049.306,255.583,-101.751,172.011,37.908,157.168
C09703=1049.312,255.832,-101.780,172.014,37.911,157.169
C09704=1049.319,256.080,-101.810,172.016,37.914,157.169
C09705=1049.325,256.329,-101.839,172.020,37.916,157.170
C09706=1049.332,256.577,-101.868,172.023,37.920,157.171
C09707=1049.339,256.825,-101.898,172.025,37.923,157.172
C09708=1049.345,257.073,-101.927,172.028,37.926,157.172
C09709=1049.351,257.321,-101.956,172.030,37.929,157.173
C09710=1049.358,257.569,-101.985,172.033,37.932,157.174
C09711=1049.365,257.817,-102.015,172.035,37.934,157.174
C09712=1049.371,258.066,-102.044,172.038,37.937,157.175
C09713=1049.377,258.314,-102.073,172.041,37.940,157.176
C09714=1049.384,258.563,-102.103,172.044,37.944,157.176
C09715=1049.391,258.810,-102.132,172.046,37.947,157.177
C09716=1049.397,259.059,-102.162,172.049,37.950,157.178
C09717=1049.404,259.307,-102.191,172.052,37.952,157.178
C09718=1049.410,259.555,-102.221,172.054,37.955,157.179
C09719=1049.417,259.803,-102.250,172.058,37.958,157.180
C09720=1049.423,260.052,-102.279,172.060,37.961,157.180
C09721=1049.430,260.299,-102.309,172.063,37.964,157.181
C09722=1049.437,260.548,-102.338,172.065,37.967,157.182
C09723=1049.444,260.796,-102.367,172.068,37.970,157.182
C09724=1049.451,261.044,-102.397,172.070,37.973,157.183
C09725=1049.457,261.292,-102.426,172.074,37.976,157.184
C09726=1049.464,261.540,-102.456,172.076,37.979,157.184
C09727=1049.471,261.788,-102.485,172.079,37.982,157.185
C09728=1049.477,262.036,-102.514,172.081,37.985,157.186
C09729=1049.484,262.285,-102.544,172.085,37.988,157.186
C09730=1049.491,262.540,-102.575,172.088,37.991,157.187
C09731=1049.497,262.794,-102.605,172.090,37.994,157.188
C09732=1049.504,263.050,-102.635,172.093,37.997,157.189
C09733=1049.511,263.305,-102.666,172.096,38.000,157.189
C09734=1049.516,263.553,-102.696,172.099,38.003,157.190
C09735=1049.523,263.801,-102.726,172.101,38.006,157.191
C09736=1049.530,264.049,-102.755,172.104,38.010,157.192
C09737=1049.536,264.297,-102.786,172.107,38.013,157.192
C09738=1049.542,264.546,-102.815,172.110,38.015,157.193
C09739=1049.549,264.794,-102.845,172.113,38.018,157.194
C09740=1049.555,265.042,-102.876,172.115,38.022,157.194
C09741=1049.562,265.290,-102.905,172.118,38.025,157.195
C09742=1049.568,265.538,-102.934,172.120,38.028,157.196
C09743=1049.575,265.786,-102.965,172.124,38.030,157.196
C09744=1049.581,266.034,-102.995,172.127,38.034,157.197
C09745=1049.588,266.283,-103.024,172.129,38.037,157.198
C09746=1049.594,266.530,-103.055,172.132,38.040,157.198
C09747=1049.601,266.779,-103.085,172.135,38.043,157.199
C09748=1049.608,267.026,-103.115,172.138,38.046,157.200
C09749=1049.614,267.275,-103.145,172.140,38.049,157.201
C09750=1049.620,267.523,-103.174,172.143,38.052,157.201
C09751=1049.627,267.771,-103.204,172.147,38.055,157.202
C09752=1049.633,268.019,-103.235,172.149,38.058,157.203
C09753=1049.640,268.267,-103.265,172.152,38.061,157.203
C09754=1049.646,268.515,-103.295,172.154,38.064,157.204
C09755=1049.653,268.764,-103.325,172.158,38.067,157.205
C09756=1049.659,269.012,-103.355,172.160,38.070,157.206
C09757=1049.666,269.260,-103.385,172.163,38.073,157.206
C09758=1049.672,269.508,-103.415,172.166,38.077,157.207
C09759=1049.679,269.756,-103.446,172.169,38.080,157.208
C09760=1049.685,270.004,-103.476,172.172,38.082,157.208
C09761=1049.692,270.252,-103.506,172.174,38.086,157.209
C09762=1049.698,270.500,-103.537,172.178,38.089,157.210
C09763=1049.705,270.748,-103.567,172.180,38.092,157.211
C09764=1049.711,270.996,-103.597,172.183,38.095,157.211
C09765=1049.718,271.244,-103.627,172.186,38.098,157.212
C09766=1049.724,271.492,-103.658,172.189,38.101,157.213
C09767=1049.731,271.740,-103.687,172.192,38.104,157.213
C09768=1049.737,271.988,-103.718,172.194,38.107,157.214
C09769=1049.744,272.237,-103.749,172.198,38.110,157.215
C09770=1049.750,272.484,-103.779,172.201,38.113,157.216
C09771=1049.757,272.733,-103.809,172.203,38.116,157.216
C09772=1049.763,272.980,-103.840,172.207,38.120,157.217
C09773=1049.770,273.228,-103.871,172.209,38.123,157.218
C09774=1049.776,273.477,-103.901,172.212,38.126,157.218
C09775=1049.782,273.725,-103.932,172.216,38.129,157.219
C09776=1049.789,273.973,-103.962,172.218,38.132,157.220
C09777=1049.795,274.221,-103.992,172.221,38.135,157.221
C09778=1049.802,274.469,-104.024,172.224,38.138,157.221
C09779=1049.809,274.717,-104.054,172.227,38.141,157.222
C09780=1049.815,274.965,-104.084,172.229,38.145,157.223
C09781=1049.821,275.213,-104.115,172.233,38.147,157.224
C09782=1049.829,275.461,-104.146,172.236,38.150,157.224
C09783=1049.835,275.709,-104.176,172.238,38.154,157.225
C09784=1049.841,275.957,-104.207,172.242,38.157,157.226
C09785=1049.848,276.205,-104.238,172.244,38.160,157.227
C09786=1049.854,276.464,-104.270,172.248,38.163,157.227
C09787=1049.861,276.724,-104.302,172.251,38.166,157.228
C09788=1049.868,276.983,-104.334,172.253,38.170,157.229
C09789=1049.874,277.242,-104.366,172.257,38.173,157.229
C09790=1049.881,277.490,-104.396,172.260,38.176,157.230
C09791=1049.888,277.738,-104.428,172.263,38.179,157.231
C09792=1049.894,277.986,-104.458,172.266,38.182,157.232
C09793=1049.901,278.234,-104.489,172.268,38.185,157.232
C09794=1049.908,278.482,-104.520,172.272,38.189,157.233
C09795=1049.914,278.731,-104.550,172.275,38.192,157.234
C09796=1049.920,278.978,-104.581,172.278,38.194,157.235
C09797=1049.927,279.226,-104.612,172.281,38.198,157.235
C09798=1049.934,279.474,-104.644,172.283,38.201,157.236
C09799=1049.940,279.723,-104.674,172.287,38.204,157.237
C09800=1049.946,279.970,-104.705,172.290,38.207,157.238
C09801=1049.953,280.218,-104.737,172.293,38.210,157.238
C09802=1049.959,280.467,-104.767,172.296,38.213,157.239
C09803=1049.966,280.714,-104.799,172.298,38.217,157.240
C09804=1049.972,280.962,-104.829,172.302,38.220,157.241
C09805=1049.979,281.210,-104.861,172.305,38.223,157.241
C09806=1049.985,281.458,-104.892,172.308,38.226,157.242
C09807=1049.992,281.707,-104.923,172.311,38.229,157.243
C09808=1049.998,281.954,-104.954,172.315,38.233,157.244
C09809=1050.005,282.202,-104.985,172.317,38.236,157.244
C09810=1050.011,282.450,-105.016,172.320,38.239,157.245
C09811=1050.018,282.698,-105.047,172.323,38.242,157.246
C09812=1050.024,282.946,-105.079,172.326,38.245,157.247
C09813=1050.031,283.193,-105.110,172.330,38.248,157.247
C09814=1050.037,283.442,-105.141,172.332,38.252,157.248
C09815=1050.044,283.690,-105.172,172.336,38.255,157.249
C09816=1050.050,283.938,-105.204,172.339,38.258,157.250
C09817=1050.057,284.185,-105.235,172.342,38.261,157.250
C09818=1050.064,284.433,-105.266,172.345,38.264,157.251
C09819=1050.070,284.681,-105.297,172.349,38.267,157.252
C09820=1050.076,284.929,-105.328,172.351,38.270,157.253
C09821=1050.083,285.177,-105.360,172.355,38.274,157.253
C09822=1050.090,285.425,-105.391,172.357,38.277,157.254
C09823=1050.097,285.673,-105.422,172.361,38.280,157.255
C09824=1050.103,285.921,-105.454,172.364,38.283,157.256
C09825=1050.110,286.169,-105.485,172.367,38.286,157.256
C09826=1050.117,286.416,-105.517,172.370,38.290,157.257
C09827=1050.123,286.664,-105.548,172.374,38.293,157.258
C09828=1050.129,286.913,-105.580,172.376,38.296,157.259
C09829=1050.136,287.161,-105.611,172.380,38.299,157.260
C09830=1050.142,287.408,-105.642,172.382,38.302,157.260
C09831=1050.149,287.656,-105.673,172.386,38.306,157.261
C09832=1050.155,287.904,-105.705,172.389,38.308,157.262
C09833=1050.162,288.151,-105.737,172.392,38.312,157.263
C09834=1050.169,288.399,-105.768,172.395,38.315,157.263
C09835=1050.175,288.648,-105.800,172.399,38.318,157.264
C09836=1050.182,288.895,-105.832,172.401,38.322,157.265
C09837=1050.189,289.143,-105.863,172.405,38.325,157.266
C09838=1050.195,289.392,-105.895,172.408,38.328,157.266
C09839=1050.201,289.639,-105.927,172.411,38.331,157.267
C09840=1050.208,289.887,-105.958,172.414,38.335,157.268
C09841=1050.215,290.135,-105.990,172.418,38.337,157.269
C09842=1050.222,290.406,-106.025,172.421,38.341,157.270
C09843=1050.229,290.676,-106.060,172.424,38.345,157.270
C09844=1050.236,290.947,-106.094,172.428,38.348,157.271
C09845=1050.243,291.218,-106.129,172.431,38.352,157.272
C09846=1050.250,291.466,-106.161,172.435,38.355,157.273
C09847=1050.257,291.713,-106.193,172.438,38.358,157.274
C09848=1050.263,291.962,-106.225,172.442,38.362,157.275
C09849=1050.270,292.210,-106.256,172.444,38.365,157.275
C09850=1050.277,292.457,-106.288,172.448,38.368,157.276
C09851=1050.283,292.705,-106.320,172.451,38.371,157.277
C09852=1050.289,292.953,-106.352,172.454,38.375,157.278
C09853=1050.296,293.201,-106.385,172.458,38.378,157.278
C09854=1050.302,293.448,-106.416,172.460,38.381,157.279
C09855=1050.309,293.696,-106.447,172.464,38.385,157.280
C09856=1050.315,293.944,-106.480,172.468,38.388,157.281
C09857=1050.322,294.192,-106.512,172.470,38.391,157.282
C09858=1050.328,294.439,-106.544,172.474,38.394,157.282
C09859=1050.336,294.688,-106.576,172.477,38.398,157.283
C09860=1050.343,294.935,-106.608,172.481,38.401,157.284
C09861=1050.349,295.184,-106.640,172.484,38.404,157.285
C09862=1050.356,295.431,-106.673,172.487,38.408,157.286
C09863=1050.362,295.679,-106.705,172.490,38.411,157.286
C09864=1050.369,295.926,-106.737,172.493,38.414,157.287
C09865=1050.375,296.175,-106.769,172.497,38.417,157.288
C09866=1050.381,296.422,-106.801,172.501,38.421,157.289
C09867=1050.388,296.669,-106.834,172.503,38.424,157.290
C09868=1050.394,296.918,-106.866,172.507,38.428,157.290
C09869=1050.401,297.166,-106.899,172.511,38.431,157.291
C09870=1050.407,297.414,-106.932,172.513,38.434,157.292
C09871=1050.413,297.662,-106.964,172.517,38.438,157.293
C09872=1050.420,297.909,-106.996,172.520,38.441,157.294
C09873=1050.427,298.157,-107.028,172.524,38.445,157.295
C09874=1050.433,298.404,-107.061,172.527,38.448,157.295
C09875=1050.439,298.652,-107.094,172.530,38.451,157.296
C09876=1050.445,298.900,-107.126,172.534,38.455,157.297
C09877=1050.452,299.147,-107.158,172.537,38.458,157.298
C09878=1050.459,299.396,-107.191,172.540,38.461,157.299
C09879=1050.465,299.643,-107.224,172.544,38.465,157.299
C09880=1050.472,299.891,-107.257,172.547,38.468,157.300
C09881=1050.478,300.139,-107.289,172.550,38.472,157.301
C09882=1050.485,300.386,-107.321,172.554,38.475,157.302
C09883=1050.491,300.634,-107.354,172.558,38.478,157.303
C09884=1050.498,300.882,-107.387,172.560,38.482,157.304
C09885=1050.504,301.130,-107.419,172.564,38.485,157.304
C09886=1050.510,301.377,-107.452,172.568,38.489,157.305
C09887=1050.517,301.625,-107.484,172.571,38.493,157.306
C09888=1050.524,301.873,-107.517,172.574,38.496,157.307
C09889=1050.531,302.121,-107.550,172.578,38.499,157.308
C09890=1050.537,302.368,-107.583,172.582,38.503,157.309
C09891=1050.543,302.616,-107.616,172.584,38.506,157.310
C09892=1050.550,302.864,-107.649,172.588,38.509,157.310
C09893=1050.557,303.111,-107.681,172.592,38.513,157.311
C09894=1050.563,303.359,-107.714,172.595,38.516,157.312
C09895=1050.570,303.606,-107.746,172.598,38.520,157.313
C09896=1050.577,303.855,-107.780,172.602,38.523,157.314
C09897=1050.583,304.102,-107.812,172.606,38.526,157.315
C09898=1050.591,304.389,-107.850,172.610,38.530,157.315
C09899=1050.598,304.675,-107.889,172.613,38.534,157.316
C09900=1050.606,304.962,-107.926,172.617,38.539,157.318
C09901=1050.614,305.249,-107.965,172.621,38.543,157.319
C09902=1050.620,305.497,-107.998,172.625,38.546,157.319
C09903=1050.627,305.745,-108.031,172.629,38.549,157.320
C09904=1050.635,305.992,-108.064,172.632,38.553,157.321
C09905=1050.641,306.240,-108.096,172.636,38.556,157.322
C09906=1050.648,306.488,-108.129,172.639,38.559,157.323
C09907=1050.654,306.735,-108.162,172.642,38.563,157.324
C09908=1050.661,306.983,-108.196,172.646,38.567,157.324
C09909=1050.668,307.231,-108.229,172.650,38.570,157.325
C09910=1050.674,307.478,-108.262,172.654,38.573,157.326
C09911=1050.681,307.726,-108.295,172.656,38.577,157.327
C09912=1050.687,307.974,-108.328,172.660,38.580,157.328
C09913=1050.695,308.222,-108.361,172.664,38.584,157.329
C09914=1050.702,308.468,-108.394,172.668,38.587,157.330
C09915=1050.708,308.717,-108.427,172.671,38.591,157.330
C09916=1050.715,308.964,-108.461,172.674,38.594,157.331
C09917=1050.722,309.212,-108.494,172.678,38.598,157.332
C09918=1050.728,309.460,-108.526,172.682,38.601,157.333
C09919=1050.735,309.707,-108.560,172.686,38.605,157.334
C09920=1050.742,309.955,-108.593,172.689,38.608,157.335
C09921=1050.749,310.203,-108.627,172.693,38.611,157.336
C09922=1050.755,310.450,-108.660,172.697,38.615,157.336
C09923=1050.762,310.698,-108.693,172.700,38.619,157.337
C09924=1050.769,310.945,-108.726,172.703,38.622,157.338
C09925=1050.777,311.193,-108.759,172.707,38.625,157.339
C09926=1050.784,311.441,-108.793,172.711,38.629,157.340
C09927=1050.790,311.688,-108.826,172.714,38.632,157.341
C09928=1050.797,311.936,-108.860,172.718,38.636,157.342
C09929=1050.804,312.183,-108.893,172.722,38.639,157.343
C09930=1050.811,312.431,-108.926,172.726,38.643,157.343
C09931=1050.818,312.679,-108.959,172.730,38.647,157.344
C09932=1050.824,312.926,-108.993,172.732,38.650,157.345
C09933=1050.832,313.174,-109.027,172.736,38.653,157.346
C09934=1050.838,313.422,-109.061,172.740,38.657,157.347
C09935=1050.844,313.670,-109.094,172.744,38.661,157.348
C09936=1050.851,313.918,-109.128,172.748,38.665,157.349
C09937=1050.857,314.164,-109.162,172.751,38.668,157.350
C09938=1050.864,314.412,-109.196,172.755,38.672,157.351
C09939=1050.870,314.659,-109.230,172.759,38.676,157.352
C09940=1050.877,314.907,-109.264,172.762,38.679,157.352
C09941=1050.883,315.154,-109.298,172.766,38.683,157.353
C09942=1050.890,315.402,-109.332,172.769,38.686,157.354
C09943=1050.897,315.650,-109.366,172.773,38.690,157.355
C09944=1050.903,315.898,-109.399,172.777,38.694,157.356
C09945=1050.910,316.146,-109.433,172.781,38.698,157.357
C09946=1050.916,316.394,-109.467,172.785,38.701,157.358
C09947=1050.923,316.641,-109.501,172.788,38.705,157.359
C09948=1050.929,316.889,-109.535,172.792,38.709,157.360
C09949=1050.936,317.135,-109.569,172.796,38.713,157.361
C09950=1050.943,317.383,-109.604,172.799,38.716,157.362
C09951=1050.950,317.631,-109.638,172.803,38.720,157.363
C09952=1050.956,317.879,-109.672,172.807,38.724,157.364
C09953=1050.963,318.126,-109.706,172.810,38.727,157.364
C09954=1050.971,318.417,-109.746,172.815,38.732,157.366
C09955=1050.979,318.708,-109.786,172.819,38.736,157.367
C09956=1050.987,318.999,-109.826,172.824,38.740,157.368
C09957=1050.995,319.290,-109.866,172.828,38.745,157.369
C09958=1051.001,319.538,-109.901,172.832,38.748,157.370
C09959=1051.008,319.785,-109.934,172.836,38.752,157.371
C09960=1051.014,320.033,-109.969,172.840,38.756,157.372
C09961=1051.022,320.280,-110.003,172.844,38.760,157.373
C09962=1051.028,320.528,-110.038,172.847,38.763,157.374
C09963=1051.035,320.776,-110.072,172.851,38.767,157.374
C09964=1051.041,321.023,-110.106,172.855,38.771,157.375
C09965=1051.048,321.271,-110.141,172.859,38.775,157.376
C09966=1051.055,321.518,-110.175,172.863,38.778,157.377
C09967=1051.062,321.766,-110.209,172.867,38.782,157.378
C09968=1051.069,322.013,-110.244,172.871,38.786,157.379
C09969=1051.076,322.261,-110.278,172.874,38.790,157.380
C09970=1051.082,322.509,-110.312,172.878,38.793,157.381
C09971=1051.090,322.756,-110.347,172.882,38.797,157.382
C09972=1051.096,323.004,-110.381,172.886,38.801,157.383
C09973=1051.103,323.251,-110.415,172.890,38.805,157.384
C09974=1051.110,323.499,-110.450,172.894,38.809,157.385
C09975=1051.116,323.746,-110.485,172.898,38.812,157.386
C09976=1051.123,323.994,-110.519,172.901,38.816,157.387
C09977=1051.130,324.241,-110.554,172.905,38.820,157.388
C09978=1051.137,324.489,-110.588,172.910,38.824,157.389
C09979=1051.144,324.736,-110.623,172.914,38.828,157.390
C09980=1051.151,324.984,-110.657,172.918,38.831,157.391
C09981=1051.158,325.231,-110.692,172.922,38.835,157.392
C09982=1051.165,325.479,-110.726,172.926,38.839,157.393
C09983=1051.172,325.726,-110.761,172.929,38.843,157.394
C09984=1051.179,325.974,-110.796,172.933,38.846,157.395
C09985=1051.185,326.222,-110.830,172.937,38.850,157.396
C09986=1051.193,326.469,-110.865,172.941,38.854,157.397
C09987=1051.200,326.716,-110.900,172.945,38.858,157.398
C09988=1051.206,326.964,-110.935,172.950,38.862,157.399
C09989=1051.214,327.211,-110.969,172.954,38.866,157.400
C09990=1051.220,327.458,-111.004,172.958,38.870,157.401
C09991=1051.227,327.707,-111.039,172.962,38.873,157.401
C09992=1051.235,327.954,-111.074,172.965,38.877,157.402
C09993=1051.242,328.201,-111.109,172.969,38.881,157.403
C09994=1051.249,328.449,-111.143,172.973,38.885,157.404
C09995=1051.256,328.696,-111.178,172.977,38.889,157.405
C09996=1051.262,328.944,-111.213,172.982,38.893,157.406
//INST
///DATE 2021/06/17 10:57
///ATTR SC,RW,RJ
////FRAME ROBOT
///GROUP1 RB1
NOP
MOVL C00000 V=800.0 PL=0
MOVL C00001 V=800.0 PL=0
MOVL C00002 V=800.0 PL=0
MOVL C00003 V=800.0 PL=0
MOVL C00004 V=800.0 PL=0
MOVL C00005 V=800.0 PL=0
MOVL C00006 V=800.0 PL=0
MOVL C00007 V=800.0 PL=0
MOVL C00008 V=800.0 PL=0
MOVL C00009 V=800.0 PL=0
MOVL C00010 V=800.0 PL=0
MOVL C00011 V=800.0 PL=0
MOVL C00012 V=800.0 PL=0
MOVL C00013 V=800.0 PL=0
MOVL C00014 V=800.0 PL=0
MOVL C00015 V=800.0 PL=0
MOVL C00016 V=800.0 PL=0
MOVL C00017 V=800.0 PL=0
MOVL C00018 V=800.0 PL=0
MOVL C00019 V=800.0 PL=0
MOVL C00020 V=800.0 PL=0
MOVL C00021 V=800.0 PL=0
MOVL C00022 V=800.0 PL=0
MOVL C00023 V=800.0 PL=0
MOVL C00024 V=800.0 PL=0
MOVL C00025 V=800.0 PL=0
MOVL C00026 V=800.0 PL=0
MOVL C00027 V=800.0 PL=0
MOVL C00028 V=800.0 PL=0
MOVL C00029 V=800.0 PL=0
MOVL C00030 V=800.0 PL=0
MOVL C00031 V=800.0 PL=0
MOVL C00032 V=800.0 PL=0
MOVL C00033 V=800.0 PL=0
MOVL C00034 V=800.0 PL=0
MOVL C00035 V=800.0 PL=0
MOVL C00036 V=800.0 PL=0
MOVL C00037 V=800.0 PL=0
MOVL C00038 V=800.0 PL=0
MOVL C00039 V=800.0 PL=0
MOVL C00040 V=800.0 PL=0
MOVL C00041 V=800.0 PL=0
MOVL C00042 V=800.0 PL=0
MOVL C00043 V=800.0 PL=0
MOVL C00044 V=800.0 PL=0
MOVL C00045 V=800.0 PL=0
MOVL C00046 V=800.0 PL=0
MOVL C00047 V=800.0 PL=0
MOVL C00048 V=800.0 PL=0
MOVL C00049 V=800.0 PL=0
MOVL C00050 V=800.0 PL=0
MOVL C00051 V=800.0 PL=0
MOVL C00052 V=800.0 PL=0
MOVL C00053 V=800.0 PL=0
MOVL C00054 V=800.0 PL=0
MOVL C00055 V=800.0 PL=0
MOVL C00056 V=800.0 PL=0
MOVL C00057 V=800.0 PL=0
MOVL C00058 V=800.0 PL=0
MOVL C00059 V=800.0 PL=0
MOVL C00060 V=800.0 PL=0
MOVL C00061 V=800.0 PL=0
MOVL C00062 V=800.0 PL=0
MOVL C00063 V=800.0 PL=0
MOVL C00064 V=800.0 PL=0
MOVL C00065 V=800.0 PL=0
MOVL C00066 V=800.0 PL=0
MOVL C00067 V=800.0 PL=0
MOVL C00068 V=800.0 PL=0
MOVL C00069 V=800.0 PL=0
MOVL C00070 V=800.0 PL=0
MOVL C00071 V=800.0 PL=0
MOVL C00072 V=800.0 PL=0
MOVL C00073 V=800.0 PL=0
MOVL C00074 V=800.0 PL=0
MOVL C00075 V=800.0 PL=0
MOVL C00076 V=800.0 PL=0
MOVL C00077 V=800.0 PL=0
MOVL C00078 V=800.0 PL=0
MOVL C00079 V=800.0 PL=0
MOVL C00080 V=800.0 PL=0
MOVL C00081 V=800.0 PL=0
MOVL C00082 V=800.0 PL=0
MOVL C00083 V=800.0 PL=0
MOVL C00084 V=800.0 PL=0
MOVL C00085 V=800.0 PL=0
MOVL C00086 V=800.0 PL=0
MOVL C00087 V=800.0 PL=0
MOVL C00088 V=800.0 PL=0
MOVL C00089 V=800.0 PL=0
MOVL C00090 V=800.0 PL=0
MOVL C00091 V=800.0 PL=0
MOVL C00092 V=800.0 PL=0
MOVL C00093 V=800.0 PL=0
MOVL C00094 V=800.0 PL=0
MOVL C00095 V=800.0 PL=0
MOVL C00096 V=800.0 PL=0
MOVL C00097 V=800.0 PL=0
MOVL C00098 V=800.0 PL=0
MOVL C00099 V=800.0 PL=0
MOVL C00100 V=800.0 PL=0
MOVL C00101 V=800.0 PL=0
MOVL C00102 V=800.0 PL=0
MOVL C00103 V=800.0 PL=0
MOVL C00104 V=800.0 PL=0
MOVL C00105 V=800.0 PL=0
MOVL C00106 V=800.0 PL=0
MOVL C00107 V=800.0 PL=0
MOVL C00108 V=800.0 PL=0
MOVL C00109 V=800.0 PL=0
MOVL C00110 V=800.0 PL=0
MOVL C00111 V=800.0 PL=0
MOVL C00112 V=800.0 PL=0
MOVL C00113 V=800.0 PL=0
MOVL C00114 V=800.0 PL=0
MOVL C00115 V=800.0 PL=0
MOVL C00116 V=800.0 PL=0
MOVL C00117 V=800.0 PL=0
MOVL C00118 V=800.0 PL=0
MOVL C00119 V=800.0 PL=0
MOVL C00120 V=800.0 PL=0
MOVL C00121 V=800.0 PL=0
MOVL C00122 V=800.0 PL=0
MOVL C00123 V=800.0 PL=0
MOVL C00124 V=800.0 PL=0
MOVL C00125 V=800.0 PL=0
MOVL C00126 V=800.0 PL=0
MOVL C00127 V=800.0 PL=0
MOVL C00128 V=800.0 PL=0
MOVL C00129 V=800.0 PL=0
MOVL C00130 V=800.0 PL=0
MOVL C00131 V=800.0 PL=0
MOVL C00132 V=800.0 PL=0
MOVL C00133 V=800.0 PL=0
MOVL C00134 V=800.0 PL=0
MOVL C00135 V=800.0 PL=0
MOVL C00136 V=800.0 PL=0
MOVL C00137 V=800.0 PL=0
MOVL C00138 V=800.0 PL=0
MOVL C00139 V=800.0 PL=0
MOVL C00140 V=800.0 PL=0
MOVL C00141 V=800.0 PL=0
MOVL C00142 V=800.0 PL=0
MOVL C00143 V=800.0 PL=0
MOVL C00144 V=800.0 PL=0
MOVL C00145 V=800.0 PL=0
MOVL C00146 V=800.0 PL=0
MOVL C00147 V=800.0 PL=0
MOVL C00148 V=800.0 PL=0
MOVL C00149 V=800.0 PL=0
MOVL C00150 V=800.0 PL=0
MOVL C00151 V=800.0 PL=0
MOVL C00152 V=800.0 PL=0
MOVL C00153 V=800.0 PL=0
MOVL C00154 V=800.0 PL=0
MOVL C00155 V=800.0 PL=0
MOVL C00156 V=800.0 PL=0
MOVL C00157 V=800.0 PL=0
MOVL C00158 V=800.0 PL=0
MOVL C00159 V=800.0 PL=0
MOVL C00160 V=800.0 PL=0
MOVL C00161 V=800.0 PL=0
MOVL C00162 V=800.0 PL=0
MOVL C00163 V=800.0 PL=0
MOVL C00164 V=800.0 PL=0
MOVL C00165 V=800.0 PL=0
MOVL C00166 V=800.0 PL=0
MOVL C00167 V=800.0 PL=0
MOVL C00168 V=800.0 PL=0
MOVL C00169 V=800.0 PL=0
MOVL C00170 V=800.0 PL=0
MOVL C00171 V=800.0 PL=0
MOVL C00172 V=800.0 PL=0
MOVL C00173 V=800.0 PL=0
MOVL C00174 V=800.0 PL=0
MOVL C00175 V=800.0 PL=0
MOVL C00176 V=800.0 PL=0
MOVL C00177 V=800.0 PL=0
MOVL C00178 V=800.0 PL=0
MOVL C00179 V=800.0 PL=0
MOVL C00180 V=800.0 PL=0
MOVL C00181 V=800.0 PL=0
MOVL C00182 V=800.0 PL=0
MOVL C00183 V=800.0 PL=0
MOVL C00184 V=800.0 PL=0
MOVL C00185 V=800.0 PL=0
MOVL C00186 V=800.0 PL=0
MOVL C00187 V=800.0 PL=0
MOVL C00188 V=800.0 PL=0
MOVL C00189 V=800.0 PL=0
MOVL C00190 V=800.0 PL=0
MOVL C00191 V=800.0 PL=0
MOVL C00192 V=800.0 PL=0
MOVL C00193 V=800.0 PL=0
MOVL C00194 V=800.0 PL=0
MOVL C00195 V=800.0 PL=0
MOVL C00196 V=800.0 PL=0
MOVL C00197 V=800.0 PL=0
MOVL C00198 V=800.0 PL=0
MOVL C00199 V=800.0 PL=0
MOVL C00200 V=800.0 PL=0
MOVL C00201 V=800.0 PL=0
MOVL C00202 V=800.0 PL=0
MOVL C00203 V=800.0 PL=0
MOVL C00204 V=800.0 PL=0
MOVL C00205 V=800.0 PL=0
MOVL C00206 V=800.0 PL=0
MOVL C00207 V=800.0 PL=0
MOVL C00208 V=800.0 PL=0
MOVL C00209 V=800.0 PL=0
MOVL C00210 V=800.0 PL=0
MOVL C00211 V=800.0 PL=0
MOVL C00212 V=800.0 PL=0
MOVL C00213 V=800.0 PL=0
MOVL C00214 V=800.0 PL=0
MOVL C00215 V=800.0 PL=0
MOVL C00216 V=800.0 PL=0
MOVL C00217 V=800.0 PL=0
MOVL C00218 V=800.0 PL=0
MOVL C00219 V=800.0 PL=0
MOVL C00220 V=800.0 PL=0
MOVL C00221 V=800.0 PL=0
MOVL C00222 V=800.0 PL=0
MOVL C00223 V=800.0 PL=0
MOVL C00224 V=800.0 PL=0
MOVL C00225 V=800.0 PL=0
MOVL C00226 V=800.0 PL=0
MOVL C00227 V=800.0 PL=0
MOVL C00228 V=800.0 PL=0
MOVL C00229 V=800.0 PL=0
MOVL C00230 V=800.0 PL=0
MOVL C00231 V=800.0 PL=0
MOVL C00232 V=800.0 PL=0
MOVL C00233 V=800.0 PL=0
MOVL C00234 V=800.0 PL=0
MOVL C00235 V=800.0 PL=0
MOVL C00236 V=800.0 PL=0
MOVL C00237 V=800.0 PL=0
MOVL C00238 V=800.0 PL=0
MOVL C00239 V=800.0 PL=0
MOVL C00240 V=800.0 PL=0
MOVL C00241 V=800.0 PL=0
MOVL C00242 V=800.0 PL=0
MOVL C00243 V=800.0 PL=0
MOVL C00244 V=800.0 PL=0
MOVL C00245 V=800.0 PL=0
MOVL C00246 V=800.0 PL=0
MOVL C00247 V=800.0 PL=0
MOVL C00248 V=800.0 PL=0
MOVL C00249 V=800.0 PL=0
MOVL C00250 V=800.0 PL=0
MOVL C00251 V=800.0 PL=0
MOVL C00252 V=800.0 PL=0
MOVL C00253 V=800.0 PL=0
MOVL C00254 V=800.0 PL=0
MOVL C00255 V=800.0 PL=0
MOVL C00256 V=800.0 PL=0
MOVL C00257 V=800.0 PL=0
MOVL C00258 V=800.0 PL=0
MOVL C00259 V=800.0 PL=0
MOVL C00260 V=800.0 PL=0
MOVL C00261 V=800.0 PL=0
MOVL C00262 V=800.0 PL=0
MOVL C00263 V=800.0 PL=0
MOVL C00264 V=800.0 PL=0
MOVL C00265 V=800.0 PL=0
MOVL C00266 V=800.0 PL=0
MOVL C00267 V=800.0 PL=0
MOVL C00268 V=800.0 PL=0
MOVL C00269 V=800.0 PL=0
MOVL C00270 V=800.0 PL=0
MOVL C00271 V=800.0 PL=0
MOVL C00272 V=800.0 PL=0
MOVL C00273 V=800.0 PL=0
MOVL C00274 V=800.0 PL=0
MOVL C00275 V=800.0 PL=0
MOVL C00276 V=800.0 PL=0
MOVL C00277 V=800.0 PL=0
MOVL C00278 V=800.0 PL=0
MOVL C00279 V=800.0 PL=0
MOVL C00280 V=800.0 PL=0
MOVL C00281 V=800.0 PL=0
MOVL C00282 V=800.0 PL=0
MOVL C00283 V=800.0 PL=0
MOVL C00284 V=800.0 PL=0
MOVL C00285 V=800.0 PL=0
MOVL C00286 V=800.0 PL=0
MOVL C00287 V=800.0 PL=0
MOVL C00288 V=800.0 PL=0
MOVL C00289 V=800.0 PL=0
MOVL C00290 V=800.0 PL=0
MOVL C00291 V=800.0 PL=0
MOVL C00292 V=800.0 PL=0
MOVL C00293 V=800.0 PL=0
MOVL C00294 V=800.0 PL=0
MOVL C00295 V=800.0 PL=0
MOVL C00296 V=800.0 PL=0
MOVL C00297 V=800.0 PL=0
MOVL C00298 V=800.0 PL=0
MOVL C00299 V=800.0 PL=0
MOVL C00300 V=800.0 PL=0
MOVL C00301 V=800.0 PL=0
MOVL C00302 V=800.0 PL=0
MOVL C00303 V=800.0 PL=0
MOVL C00304 V=800.0 PL=0
MOVL C00305 V=800.0 PL=0
MOVL C00306 V=800.0 PL=0
MOVL C00307 V=800.0 PL=0
MOVL C00308 V=800.0 PL=0
MOVL C00309 V=800.0 PL=0
MOVL C00310 V=800.0 PL=0
MOVL C00311 V=800.0 PL=0
MOVL C00312 V=800.0 PL=0
MOVL C00313 V=800.0 PL=0
MOVL C00314 V=800.0 PL=0
MOVL C00315 V=800.0 PL=0
MOVL C00316 V=800.0 PL=0
MOVL C00317 V=800.0 PL=0
MOVL C00318 V=800.0 PL=0
MOVL C00319 V=800.0 PL=0
MOVL C00320 V=800.0 PL=0
MOVL C00321 V=800.0 PL=0
MOVL C00322 V=800.0 PL=0
MOVL C00323 V=800.0 PL=0
MOVL C00324 V=800.0 PL=0
MOVL C00325 V=800.0 PL=0
MOVL C00326 V=800.0 PL=0
MOVL C00327 V=800.0 PL=0
MOVL C00328 V=800.0 PL=0
MOVL C00329 V=800.0 PL=0
MOVL C00330 V=800.0 PL=0
MOVL C00331 V=800.0 PL=0
MOVL C00332 V=800.0 PL=0
MOVL C00333 V=800.0 PL=0
MOVL C00334 V=800.0 PL=0
MOVL C00335 V=800.0 PL=0
MOVL C00336 V=800.0 PL=0
MOVL C00337 V=800.0 PL=0
MOVL C00338 V=800.0 PL=0
MOVL C00339 V=800.0 PL=0
MOVL C00340 V=800.0 PL=0
MOVL C00341 V=800.0 PL=0
MOVL C00342 V=800.0 PL=0
MOVL C00343 V=800.0 PL=0
MOVL C00344 V=800.0 PL=0
MOVL C00345 V=800.0 PL=0
MOVL C00346 V=800.0 PL=0
MOVL C00347 V=800.0 PL=0
MOVL C00348 V=800.0 PL=0
MOVL C00349 V=800.0 PL=0
MOVL C00350 V=800.0 PL=0
MOVL C00351 V=800.0 PL=0
MOVL C00352 V=800.0 PL=0
MOVL C00353 V=800.0 PL=0
MOVL C00354 V=800.0 PL=0
MOVL C00355 V=800.0 PL=0
MOVL C00356 V=800.0 PL=0
MOVL C00357 V=800.0 PL=0
MOVL C00358 V=800.0 PL=0
MOVL C00359 V=800.0 PL=0
MOVL C00360 V=800.0 PL=0
MOVL C00361 V=800.0 PL=0
MOVL C00362 V=800.0 PL=0
MOVL C00363 V=800.0 PL=0
MOVL C00364 V=800.0 PL=0
MOVL C00365 V=800.0 PL=0
MOVL C00366 V=800.0 PL=0
MOVL C00367 V=800.0 PL=0
MOVL C00368 V=800.0 PL=0
MOVL C00369 V=800.0 PL=0
MOVL C00370 V=800.0 PL=0
MOVL C00371 V=800.0 PL=0
MOVL C00372 V=800.0 PL=0
MOVL C00373 V=800.0 PL=0
MOVL C00374 V=800.0 PL=0
MOVL C00375 V=800.0 PL=0
MOVL C00376 V=800.0 PL=0
MOVL C00377 V=800.0 PL=0
MOVL C00378 V=800.0 PL=0
MOVL C00379 V=800.0 PL=0
MOVL C00380 V=800.0 PL=0
MOVL C00381 V=800.0 PL=0
MOVL C00382 V=800.0 PL=0
MOVL C00383 V=800.0 PL=0
MOVL C00384 V=800.0 PL=0
MOVL C00385 V=800.0 PL=0
MOVL C00386 V=800.0 PL=0
MOVL C00387 V=800.0 PL=0
MOVL C00388 V=800.0 PL=0
MOVL C00389 V=800.0 PL=0
MOVL C00390 V=800.0 PL=0
MOVL C00391 V=800.0 PL=0
MOVL C00392 V=800.0 PL=0
MOVL C00393 V=800.0 PL=0
MOVL C00394 V=800.0 PL=0
MOVL C00395 V=800.0 PL=0
MOVL C00396 V=800.0 PL=0
MOVL C00397 V=800.0 PL=0
MOVL C00398 V=800.0 PL=0
MOVL C00399 V=800.0 PL=0
MOVL C00400 V=800.0 PL=0
MOVL C00401 V=800.0 PL=0
MOVL C00402 V=800.0 PL=0
MOVL C00403 V=800.0 PL=0
MOVL C00404 V=800.0 PL=0
MOVL C00405 V=800.0 PL=0
MOVL C00406 V=800.0 PL=0
MOVL C00407 V=800.0 PL=0
MOVL C00408 V=800.0 PL=0
MOVL C00409 V=800.0 PL=0
MOVL C00410 V=800.0 PL=0
MOVL C00411 V=800.0 PL=0
MOVL C00412 V=800.0 PL=0
MOVL C00413 V=800.0 PL=0
MOVL C00414 V=800.0 PL=0
MOVL C00415 V=800.0 PL=0
MOVL C00416 V=800.0 PL=0
MOVL C00417 V=800.0 PL=0
MOVL C00418 V=800.0 PL=0
MOVL C00419 V=800.0 PL=0
MOVL C00420 V=800.0 PL=0
MOVL C00421 V=800.0 PL=0
MOVL C00422 V=800.0 PL=0
MOVL C00423 V=800.0 PL=0
MOVL C00424 V=800.0 PL=0
MOVL C00425 V=800.0 PL=0
MOVL C00426 V=800.0 PL=0
MOVL C00427 V=800.0 PL=0
MOVL C00428 V=800.0 PL=0
MOVL C00429 V=800.0 PL=0
MOVL C00430 V=800.0 PL=0
MOVL C00431 V=800.0 PL=0
MOVL C00432 V=800.0 PL=0
MOVL C00433 V=800.0 PL=0
MOVL C00434 V=800.0 PL=0
MOVL C00435 V=800.0 PL=0
MOVL C00436 V=800.0 PL=0
MOVL C00437 V=800.0 PL=0
MOVL C00438 V=800.0 PL=0
MOVL C00439 V=800.0 PL=0
MOVL C00440 V=800.0 PL=0
MOVL C00441 V=800.0 PL=0
MOVL C00442 V=800.0 PL=0
MOVL C00443 V=800.0 PL=0
MOVL C00444 V=800.0 PL=0
MOVL C00445 V=800.0 PL=0
MOVL C00446 V=800.0 PL=0
MOVL C00447 V=800.0 PL=0
MOVL C00448 V=800.0 PL=0
MOVL C00449 V=800.0 PL=0
MOVL C00450 V=800.0 PL=0
MOVL C00451 V=800.0 PL=0
MOVL C00452 V=800.0 PL=0
MOVL C00453 V=800.0 PL=0
MOVL C00454 V=800.0 PL=0
MOVL C00455 V=800.0 PL=0
MOVL C00456 V=800.0 PL=0
MOVL C00457 V=800.0 PL=0
MOVL C00458 V=800.0 PL=0
MOVL C00459 V=800.0 PL=0
MOVL C00460 V=800.0 PL=0
MOVL C00461 V=800.0 PL=0
MOVL C00462 V=800.0 PL=0
MOVL C00463 V=800.0 PL=0
MOVL C00464 V=800.0 PL=0
MOVL C00465 V=800.0 PL=0
MOVL C00466 V=800.0 PL=0
MOVL C00467 V=800.0 PL=0
MOVL C00468 V=800.0 PL=0
MOVL C00469 V=800.0 PL=0
MOVL C00470 V=800.0 PL=0
MOVL C00471 V=800.0 PL=0
MOVL C00472 V=800.0 PL=0
MOVL C00473 V=800.0 PL=0
MOVL C00474 V=800.0 PL=0
MOVL C00475 V=800.0 PL=0
MOVL C00476 V=800.0 PL=0
MOVL C00477 V=800.0 PL=0
MOVL C00478 V=800.0 PL=0
MOVL C00479 V=800.0 PL=0
MOVL C00480 V=800.0 PL=0
MOVL C00481 V=800.0 PL=0
MOVL C00482 V=800.0 PL=0
MOVL C00483 V=800.0 PL=0
MOVL C00484 V=800.0 PL=0
MOVL C00485 V=800.0 PL=0
MOVL C00486 V=800.0 PL=0
MOVL C00487 V=800.0 PL=0
MOVL C00488 V=800.0 PL=0
MOVL C00489 V=800.0 PL=0
MOVL C00490 V=800.0 PL=0
MOVL C00491 V=800.0 PL=0
MOVL C00492 V=800.0 PL=0
MOVL C00493 V=800.0 PL=0
MOVL C00494 V=800.0 PL=0
MOVL C00495 V=800.0 PL=0
MOVL C00496 V=800.0 PL=0
MOVL C00497 V=800.0 PL=0
MOVL C00498 V=800.0 PL=0
MOVL C00499 V=800.0 PL=0
MOVL C00500 V=800.0 PL=0
MOVL C00501 V=800.0 PL=0
MOVL C00502 V=800.0 PL=0
MOVL C00503 V=800.0 PL=0
MOVL C00504 V=800.0 PL=0
MOVL C00505 V=800.0 PL=0
MOVL C00506 V=800.0 PL=0
MOVL C00507 V=800.0 PL=0
MOVL C00508 V=800.0 PL=0
MOVL C00509 V=800.0 PL=0
MOVL C00510 V=800.0 PL=0
MOVL C00511 V=800.0 PL=0
MOVL C00512 V=800.0 PL=0
MOVL C00513 V=800.0 PL=0
MOVL C00514 V=800.0 PL=0
MOVL C00515 V=800.0 PL=0
MOVL C00516 V=800.0 PL=0
MOVL C00517 V=800.0 PL=0
MOVL C00518 V=800.0 PL=0
MOVL C00519 V=800.0 PL=0
MOVL C00520 V=800.0 PL=0
MOVL C00521 V=800.0 PL=0
MOVL C00522 V=800.0 PL=0
MOVL C00523 V=800.0 PL=0
MOVL C00524 V=800.0 PL=0
MOVL C00525 V=800.0 PL=0
MOVL C00526 V=800.0 PL=0
MOVL C00527 V=800.0 PL=0
MOVL C00528 V=800.0 PL=0
MOVL C00529 V=800.0 PL=0
MOVL C00530 V=800.0 PL=0
MOVL C00531 V=800.0 PL=0
MOVL C00532 V=800.0 PL=0
MOVL C00533 V=800.0 PL=0
MOVL C00534 V=800.0 PL=0
MOVL C00535 V=800.0 PL=0
MOVL C00536 V=800.0 PL=0
MOVL C00537 V=800.0 PL=0
MOVL C00538 V=800.0 PL=0
MOVL C00539 V=800.0 PL=0
MOVL C00540 V=800.0 PL=0
MOVL C00541 V=800.0 PL=0
MOVL C00542 V=800.0 PL=0
MOVL C00543 V=800.0 PL=0
MOVL C00544 V=800.0 PL=0
MOVL C00545 V=800.0 PL=0
MOVL C00546 V=800.0 PL=0
MOVL C00547 V=800.0 PL=0
MOVL C00548 V=800.0 PL=0
MOVL C00549 V=800.0 PL=0
MOVL C00550 V=800.0 PL=0
MOVL C00551 V=800.0 PL=0
MOVL C00552 V=800.0 PL=0
MOVL C00553 V=800.0 PL=0
MOVL C00554 V=800.0 PL=0
MOVL C00555 V=800.0 PL=0
MOVL C00556 V=800.0 PL=0
MOVL C00557 V=800.0 PL=0
MOVL C00558 V=800.0 PL=0
MOVL C00559 V=800.0 PL=0
MOVL C00560 V=800.0 PL=0
MOVL C00561 V=800.0 PL=0
MOVL C00562 V=800.0 PL=0
MOVL C00563 V=800.0 PL=0
MOVL C00564 V=800.0 PL=0
MOVL C00565 V=800.0 PL=0
MOVL C00566 V=800.0 PL=0
MOVL C00567 V=800.0 PL=0
MOVL C00568 V=800.0 PL=0
MOVL C00569 V=800.0 PL=0
MOVL C00570 V=800.0 PL=0
MOVL C00571 V=800.0 PL=0
MOVL C00572 V=800.0 PL=0
MOVL C00573 V=800.0 PL=0
MOVL C00574 V=800.0 PL=0
MOVL C00575 V=800.0 PL=0
MOVL C00576 V=800.0 PL=0
MOVL C00577 V=800.0 PL=0
MOVL C00578 V=800.0 PL=0
MOVL C00579 V=800.0 PL=0
MOVL C00580 V=800.0 PL=0
MOVL C00581 V=800.0 PL=0
MOVL C00582 V=800.0 PL=0
MOVL C00583 V=800.0 PL=0
MOVL C00584 V=800.0 PL=0
MOVL C00585 V=800.0 PL=0
MOVL C00586 V=800.0 PL=0
MOVL C00587 V=800.0 PL=0
MOVL C00588 V=800.0 PL=0
MOVL C00589 V=800.0 PL=0
MOVL C00590 V=800.0 PL=0
MOVL C00591 V=800.0 PL=0
MOVL C00592 V=800.0 PL=0
MOVL C00593 V=800.0 PL=0
MOVL C00594 V=800.0 PL=0
MOVL C00595 V=800.0 PL=0
MOVL C00596 V=800.0 PL=0
MOVL C00597 V=800.0 PL=0
MOVL C00598 V=800.0 PL=0
MOVL C00599 V=800.0 PL=0
MOVL C00600 V=800.0 PL=0
MOVL C00601 V=800.0 PL=0
MOVL C00602 V=800.0 PL=0
MOVL C00603 V=800.0 PL=0
MOVL C00604 V=800.0 PL=0
MOVL C00605 V=800.0 PL=0
MOVL C00606 V=800.0 PL=0
MOVL C00607 V=800.0 PL=0
MOVL C00608 V=800.0 PL=0
MOVL C00609 V=800.0 PL=0
MOVL C00610 V=800.0 PL=0
MOVL C00611 V=800.0 PL=0
MOVL C00612 V=800.0 PL=0
MOVL C00613 V=800.0 PL=0
MOVL C00614 V=800.0 PL=0
MOVL C00615 V=800.0 PL=0
MOVL C00616 V=800.0 PL=0
MOVL C00617 V=800.0 PL=0
MOVL C00618 V=800.0 PL=0
MOVL C00619 V=800.0 PL=0
MOVL C00620 V=800.0 PL=0
MOVL C00621 V=800.0 PL=0
MOVL C00622 V=800.0 PL=0
MOVL C00623 V=800.0 PL=0
MOVL C00624 V=800.0 PL=0
MOVL C00625 V=800.0 PL=0
MOVL C00626 V=800.0 PL=0
MOVL C00627 V=800.0 PL=0
MOVL C00628 V=800.0 PL=0
MOVL C00629 V=800.0 PL=0
MOVL C00630 V=800.0 PL=0
MOVL C00631 V=800.0 PL=0
MOVL C00632 V=800.0 PL=0
MOVL C00633 V=800.0 PL=0
MOVL C00634 V=800.0 PL=0
MOVL C00635 V=800.0 PL=0
MOVL C00636 V=800.0 PL=0
MOVL C00637 V=800.0 PL=0
MOVL C00638 V=800.0 PL=0
MOVL C00639 V=800.0 PL=0
MOVL C00640 V=800.0 PL=0
MOVL C00641 V=800.0 PL=0
MOVL C00642 V=800.0 PL=0
MOVL C00643 V=800.0 PL=0
MOVL C00644 V=800.0 PL=0
MOVL C00645 V=800.0 PL=0
MOVL C00646 V=800.0 PL=0
MOVL C00647 V=800.0 PL=0
MOVL C00648 V=800.0 PL=0
MOVL C00649 V=800.0 PL=0
MOVL C00650 V=800.0 PL=0
MOVL C00651 V=800.0 PL=0
MOVL C00652 V=800.0 PL=0
MOVL C00653 V=800.0 PL=0
MOVL C00654 V=800.0 PL=0
MOVL C00655 V=800.0 PL=0
MOVL C00656 V=800.0 PL=0
MOVL C00657 V=800.0 PL=0
MOVL C00658 V=800.0 PL=0
MOVL C00659 V=800.0 PL=0
MOVL C00660 V=800.0 PL=0
MOVL C00661 V=800.0 PL=0
MOVL C00662 V=800.0 PL=0
MOVL C00663 V=800.0 PL=0
MOVL C00664 V=800.0 PL=0
MOVL C00665 V=800.0 PL=0
MOVL C00666 V=800.0 PL=0
MOVL C00667 V=800.0 PL=0
MOVL C00668 V=800.0 PL=0
MOVL C00669 V=800.0 PL=0
MOVL C00670 V=800.0 PL=0
MOVL C00671 V=800.0 PL=0
MOVL C00672 V=800.0 PL=0
MOVL C00673 V=800.0 PL=0
MOVL C00674 V=800.0 PL=0
MOVL C00675 V=800.0 PL=0
MOVL C00676 V=800.0 PL=0
MOVL C00677 V=800.0 PL=0
MOVL C00678 V=800.0 PL=0
MOVL C00679 V=800.0 PL=0
MOVL C00680 V=800.0 PL=0
MOVL C00681 V=800.0 PL=0
MOVL C00682 V=800.0 PL=0
MOVL C00683 V=800.0 PL=0
MOVL C00684 V=800.0 PL=0
MOVL C00685 V=800.0 PL=0
MOVL C00686 V=800.0 PL=0
MOVL C00687 V=800.0 PL=0
MOVL C00688 V=800.0 PL=0
MOVL C00689 V=800.0 PL=0
MOVL C00690 V=800.0 PL=0
MOVL C00691 V=800.0 PL=0
MOVL C00692 V=800.0 PL=0
MOVL C00693 V=800.0 PL=0
MOVL C00694 V=800.0 PL=0
MOVL C00695 V=800.0 PL=0
MOVL C00696 V=800.0 PL=0
MOVL C00697 V=800.0 PL=0
MOVL C00698 V=800.0 PL=0
MOVL C00699 V=800.0 PL=0
MOVL C00700 V=800.0 PL=0
MOVL C00701 V=800.0 PL=0
MOVL C00702 V=800.0 PL=0
MOVL C00703 V=800.0 PL=0
MOVL C00704 V=800.0 PL=0
MOVL C00705 V=800.0 PL=0
MOVL C00706 V=800.0 PL=0
MOVL C00707 V=800.0 PL=0
MOVL C00708 V=800.0 PL=0
MOVL C00709 V=800.0 PL=0
MOVL C00710 V=800.0 PL=0
MOVL C00711 V=800.0 PL=0
MOVL C00712 V=800.0 PL=0
MOVL C00713 V=800.0 PL=0
MOVL C00714 V=800.0 PL=0
MOVL C00715 V=800.0 PL=0
MOVL C00716 V=800.0 PL=0
MOVL C00717 V=800.0 PL=0
MOVL C00718 V=800.0 PL=0
MOVL C00719 V=800.0 PL=0
MOVL C00720 V=800.0 PL=0
MOVL C00721 V=800.0 PL=0
MOVL C00722 V=800.0 PL=0
MOVL C00723 V=800.0 PL=0
MOVL C00724 V=800.0 PL=0
MOVL C00725 V=800.0 PL=0
MOVL C00726 V=800.0 PL=0
MOVL C00727 V=800.0 PL=0
MOVL C00728 V=800.0 PL=0
MOVL C00729 V=800.0 PL=0
MOVL C00730 V=800.0 PL=0
MOVL C00731 V=800.0 PL=0
MOVL C00732 V=800.0 PL=0
MOVL C00733 V=800.0 PL=0
MOVL C00734 V=800.0 PL=0
MOVL C00735 V=800.0 PL=0
MOVL C00736 V=800.0 PL=0
MOVL C00737 V=800.0 PL=0
MOVL C00738 V=800.0 PL=0
MOVL C00739 V=800.0 PL=0
MOVL C00740 V=800.0 PL=0
MOVL C00741 V=800.0 PL=0
MOVL C00742 V=800.0 PL=0
MOVL C00743 V=800.0 PL=0
MOVL C00744 V=800.0 PL=0
MOVL C00745 V=800.0 PL=0
MOVL C00746 V=800.0 PL=0
MOVL C00747 V=800.0 PL=0
MOVL C00748 V=800.0 PL=0
MOVL C00749 V=800.0 PL=0
MOVL C00750 V=800.0 PL=0
MOVL C00751 V=800.0 PL=0
MOVL C00752 V=800.0 PL=0
MOVL C00753 V=800.0 PL=0
MOVL C00754 V=800.0 PL=0
MOVL C00755 V=800.0 PL=0
MOVL C00756 V=800.0 PL=0
MOVL C00757 V=800.0 PL=0
MOVL C00758 V=800.0 PL=0
MOVL C00759 V=800.0 PL=0
MOVL C00760 V=800.0 PL=0
MOVL C00761 V=800.0 PL=0
MOVL C00762 V=800.0 PL=0
MOVL C00763 V=800.0 PL=0
MOVL C00764 V=800.0 PL=0
MOVL C00765 V=800.0 PL=0
MOVL C00766 V=800.0 PL=0
MOVL C00767 V=800.0 PL=0
MOVL C00768 V=800.0 PL=0
MOVL C00769 V=800.0 PL=0
MOVL C00770 V=800.0 PL=0
MOVL C00771 V=800.0 PL=0
MOVL C00772 V=800.0 PL=0
MOVL C00773 V=800.0 PL=0
MOVL C00774 V=800.0 PL=0
MOVL C00775 V=800.0 PL=0
MOVL C00776 V=800.0 PL=0
MOVL C00777 V=800.0 PL=0
MOVL C00778 V=800.0 PL=0
MOVL C00779 V=800.0 PL=0
MOVL C00780 V=800.0 PL=0
MOVL C00781 V=800.0 PL=0
MOVL C00782 V=800.0 PL=0
MOVL C00783 V=800.0 PL=0
MOVL C00784 V=800.0 PL=0
MOVL C00785 V=800.0 PL=0
MOVL C00786 V=800.0 PL=0
MOVL C00787 V=800.0 PL=0
MOVL C00788 V=800.0 PL=0
MOVL C00789 V=800.0 PL=0
MOVL C00790 V=800.0 PL=0
MOVL C00791 V=800.0 PL=0
MOVL C00792 V=800.0 PL=0
MOVL C00793 V=800.0 PL=0
MOVL C00794 V=800.0 PL=0
MOVL C00795 V=800.0 PL=0
MOVL C00796 V=800.0 PL=0
MOVL C00797 V=800.0 PL=0
MOVL C00798 V=800.0 PL=0
MOVL C00799 V=800.0 PL=0
MOVL C00800 V=800.0 PL=0
MOVL C00801 V=800.0 PL=0
MOVL C00802 V=800.0 PL=0
MOVL C00803 V=800.0 PL=0
MOVL C00804 V=800.0 PL=0
MOVL C00805 V=800.0 PL=0
MOVL C00806 V=800.0 PL=0
MOVL C00807 V=800.0 PL=0
MOVL C00808 V=800.0 PL=0
MOVL C00809 V=800.0 PL=0
MOVL C00810 V=800.0 PL=0
MOVL C00811 V=800.0 PL=0
MOVL C00812 V=800.0 PL=0
MOVL C00813 V=800.0 PL=0
MOVL C00814 V=800.0 PL=0
MOVL C00815 V=800.0 PL=0
MOVL C00816 V=800.0 PL=0
MOVL C00817 V=800.0 PL=0
MOVL C00818 V=800.0 PL=0
MOVL C00819 V=800.0 PL=0
MOVL C00820 V=800.0 PL=0
MOVL C00821 V=800.0 PL=0
MOVL C00822 V=800.0 PL=0
MOVL C00823 V=800.0 PL=0
MOVL C00824 V=800.0 PL=0
MOVL C00825 V=800.0 PL=0
MOVL C00826 V=800.0 PL=0
MOVL C00827 V=800.0 PL=0
MOVL C00828 V=800.0 PL=0
MOVL C00829 V=800.0 PL=0
MOVL C00830 V=800.0 PL=0
MOVL C00831 V=800.0 PL=0
MOVL C00832 V=800.0 PL=0
MOVL C00833 V=800.0 PL=0
MOVL C00834 V=800.0 PL=0
MOVL C00835 V=800.0 PL=0
MOVL C00836 V=800.0 PL=0
MOVL C00837 V=800.0 PL=0
MOVL C00838 V=800.0 PL=0
MOVL C00839 V=800.0 PL=0
MOVL C00840 V=800.0 PL=0
MOVL C00841 V=800.0 PL=0
MOVL C00842 V=800.0 PL=0
MOVL C00843 V=800.0 PL=0
MOVL C00844 V=800.0 PL=0
MOVL C00845 V=800.0 PL=0
MOVL C00846 V=800.0 PL=0
MOVL C00847 V=800.0 PL=0
MOVL C00848 V=800.0 PL=0
MOVL C00849 V=800.0 PL=0
MOVL C00850 V=800.0 PL=0
MOVL C00851 V=800.0 PL=0
MOVL C00852 V=800.0 PL=0
MOVL C00853 V=800.0 PL=0
MOVL C00854 V=800.0 PL=0
MOVL C00855 V=800.0 PL=0
MOVL C00856 V=800.0 PL=0
MOVL C00857 V=800.0 PL=0
MOVL C00858 V=800.0 PL=0
MOVL C00859 V=800.0 PL=0
MOVL C00860 V=800.0 PL=0
MOVL C00861 V=800.0 PL=0
MOVL C00862 V=800.0 PL=0
MOVL C00863 V=800.0 PL=0
MOVL C00864 V=800.0 PL=0
MOVL C00865 V=800.0 PL=0
MOVL C00866 V=800.0 PL=0
MOVL C00867 V=800.0 PL=0
MOVL C00868 V=800.0 PL=0
MOVL C00869 V=800.0 PL=0
MOVL C00870 V=800.0 PL=0
MOVL C00871 V=800.0 PL=0
MOVL C00872 V=800.0 PL=0
MOVL C00873 V=800.0 PL=0
MOVL C00874 V=800.0 PL=0
MOVL C00875 V=800.0 PL=0
MOVL C00876 V=800.0 PL=0
MOVL C00877 V=800.0 PL=0
MOVL C00878 V=800.0 PL=0
MOVL C00879 V=800.0 PL=0
MOVL C00880 V=800.0 PL=0
MOVL C00881 V=800.0 PL=0
MOVL C00882 V=800.0 PL=0
MOVL C00883 V=800.0 PL=0
MOVL C00884 V=800.0 PL=0
MOVL C00885 V=800.0 PL=0
MOVL C00886 V=800.0 PL=0
MOVL C00887 V=800.0 PL=0
MOVL C00888 V=800.0 PL=0
MOVL C00889 V=800.0 PL=0
MOVL C00890 V=800.0 PL=0
MOVL C00891 V=800.0 PL=0
MOVL C00892 V=800.0 PL=0
MOVL C00893 V=800.0 PL=0
MOVL C00894 V=800.0 PL=0
MOVL C00895 V=800.0 PL=0
MOVL C00896 V=800.0 PL=0
MOVL C00897 V=800.0 PL=0
MOVL C00898 V=800.0 PL=0
MOVL C00899 V=800.0 PL=0
MOVL C00900 V=800.0 PL=0
MOVL C00901 V=800.0 PL=0
MOVL C00902 V=800.0 PL=0
MOVL C00903 V=800.0 PL=0
MOVL C00904 V=800.0 PL=0
MOVL C00905 V=800.0 PL=0
MOVL C00906 V=800.0 PL=0
MOVL C00907 V=800.0 PL=0
MOVL C00908 V=800.0 PL=0
MOVL C00909 V=800.0 PL=0
MOVL C00910 V=800.0 PL=0
MOVL C00911 V=800.0 PL=0
MOVL C00912 V=800.0 PL=0
MOVL C00913 V=800.0 PL=0
MOVL C00914 V=800.0 PL=0
MOVL C00915 V=800.0 PL=0
MOVL C00916 V=800.0 PL=0
MOVL C00917 V=800.0 PL=0
MOVL C00918 V=800.0 PL=0
MOVL C00919 V=800.0 PL=0
MOVL C00920 V=800.0 PL=0
MOVL C00921 V=800.0 PL=0
MOVL C00922 V=800.0 PL=0
MOVL C00923 V=800.0 PL=0
MOVL C00924 V=800.0 PL=0
MOVL C00925 V=800.0 PL=0
MOVL C00926 V=800.0 PL=0
MOVL C00927 V=800.0 PL=0
MOVL C00928 V=800.0 PL=0
MOVL C00929 V=800.0 PL=0
MOVL C00930 V=800.0 PL=0
MOVL C00931 V=800.0 PL=0
MOVL C00932 V=800.0 PL=0
MOVL C00933 V=800.0 PL=0
MOVL C00934 V=800.0 PL=0
MOVL C00935 V=800.0 PL=0
MOVL C00936 V=800.0 PL=0
MOVL C00937 V=800.0 PL=0
MOVL C00938 V=800.0 PL=0
MOVL C00939 V=800.0 PL=0
MOVL C00940 V=800.0 PL=0
MOVL C00941 V=800.0 PL=0
MOVL C00942 V=800.0 PL=0
MOVL C00943 V=800.0 PL=0
MOVL C00944 V=800.0 PL=0
MOVL C00945 V=800.0 PL=0
MOVL C00946 V=800.0 PL=0
MOVL C00947 V=800.0 PL=0
MOVL C00948 V=800.0 PL=0
MOVL C00949 V=800.0 PL=0
MOVL C00950 V=800.0 PL=0
MOVL C00951 V=800.0 PL=0
MOVL C00952 V=800.0 PL=0
MOVL C00953 V=800.0 PL=0
MOVL C00954 V=800.0 PL=0
MOVL C00955 V=800.0 PL=0
MOVL C00956 V=800.0 PL=0
MOVL C00957 V=800.0 PL=0
MOVL C00958 V=800.0 PL=0
MOVL C00959 V=800.0 PL=0
MOVL C00960 V=800.0 PL=0
MOVL C00961 V=800.0 PL=0
MOVL C00962 V=800.0 PL=0
MOVL C00963 V=800.0 PL=0
MOVL C00964 V=800.0 PL=0
MOVL C00965 V=800.0 PL=0
MOVL C00966 V=800.0 PL=0
MOVL C00967 V=800.0 PL=0
MOVL C00968 V=800.0 PL=0
MOVL C00969 V=800.0 PL=0
MOVL C00970 V=800.0 PL=0
MOVL C00971 V=800.0 PL=0
MOVL C00972 V=800.0 PL=0
MOVL C00973 V=800.0 PL=0
MOVL C00974 V=800.0 PL=0
MOVL C00975 V=800.0 PL=0
MOVL C00976 V=800.0 PL=0
MOVL C00977 V=800.0 PL=0
MOVL C00978 V=800.0 PL=0
MOVL C00979 V=800.0 PL=0
MOVL C00980 V=800.0 PL=0
MOVL C00981 V=800.0 PL=0
MOVL C00982 V=800.0 PL=0
MOVL C00983 V=800.0 PL=0
MOVL C00984 V=800.0 PL=0
MOVL C00985 V=800.0 PL=0
MOVL C00986 V=800.0 PL=0
MOVL C00987 V=800.0 PL=0
MOVL C00988 V=800.0 PL=0
MOVL C00989 V=800.0 PL=0
MOVL C00990 V=800.0 PL=0
MOVL C00991 V=800.0 PL=0
MOVL C00992 V=800.0 PL=0
MOVL C00993 V=800.0 PL=0
MOVL C00994 V=800.0 PL=0
MOVL C00995 V=800.0 PL=0
MOVL C00996 V=800.0 PL=0
MOVL C00997 V=800.0 PL=0
MOVL C00998 V=800.0 PL=0
MOVL C00999 V=800.0 PL=0
MOVL C01000 V=800.0 PL=0
MOVL C01001 V=800.0 PL=0
MOVL C01002 V=800.0 PL=0
MOVL C01003 V=800.0 PL=0
MOVL C01004 V=800.0 PL=0
MOVL C01005 V=800.0 PL=0
MOVL C01006 V=800.0 PL=0
MOVL C01007 V=800.0 PL=0
MOVL C01008 V=800.0 PL=0
MOVL C01009 V=800.0 PL=0
MOVL C01010 V=800.0 PL=0
MOVL C01011 V=800.0 PL=0
MOVL C01012 V=800.0 PL=0
MOVL C01013 V=800.0 PL=0
MOVL C01014 V=800.0 PL=0
MOVL C01015 V=800.0 PL=0
MOVL C01016 V=800.0 PL=0
MOVL C01017 V=800.0 PL=0
MOVL C01018 V=800.0 PL=0
MOVL C01019 V=800.0 PL=0
MOVL C01020 V=800.0 PL=0
MOVL C01021 V=800.0 PL=0
MOVL C01022 V=800.0 PL=0
MOVL C01023 V=800.0 PL=0
MOVL C01024 V=800.0 PL=0
MOVL C01025 V=800.0 PL=0
MOVL C01026 V=800.0 PL=0
MOVL C01027 V=800.0 PL=0
MOVL C01028 V=800.0 PL=0
MOVL C01029 V=800.0 PL=0
MOVL C01030 V=800.0 PL=0
MOVL C01031 V=800.0 PL=0
MOVL C01032 V=800.0 PL=0
MOVL C01033 V=800.0 PL=0
MOVL C01034 V=800.0 PL=0
MOVL C01035 V=800.0 PL=0
MOVL C01036 V=800.0 PL=0
MOVL C01037 V=800.0 PL=0
MOVL C01038 V=800.0 PL=0
MOVL C01039 V=800.0 PL=0
MOVL C01040 V=800.0 PL=0
MOVL C01041 V=800.0 PL=0
MOVL C01042 V=800.0 PL=0
MOVL C01043 V=800.0 PL=0
MOVL C01044 V=800.0 PL=0
MOVL C01045 V=800.0 PL=0
MOVL C01046 V=800.0 PL=0
MOVL C01047 V=800.0 PL=0
MOVL C01048 V=800.0 PL=0
MOVL C01049 V=800.0 PL=0
MOVL C01050 V=800.0 PL=0
MOVL C01051 V=800.0 PL=0
MOVL C01052 V=800.0 PL=0
MOVL C01053 V=800.0 PL=0
MOVL C01054 V=800.0 PL=0
MOVL C01055 V=800.0 PL=0
MOVL C01056 V=800.0 PL=0
MOVL C01057 V=800.0 PL=0
MOVL C01058 V=800.0 PL=0
MOVL C01059 V=800.0 PL=0
MOVL C01060 V=800.0 PL=0
MOVL C01061 V=800.0 PL=0
MOVL C01062 V=800.0 PL=0
MOVL C01063 V=800.0 PL=0
MOVL C01064 V=800.0 PL=0
MOVL C01065 V=800.0 PL=0
MOVL C01066 V=800.0 PL=0
MOVL C01067 V=800.0 PL=0
MOVL C01068 V=800.0 PL=0
MOVL C01069 V=800.0 PL=0
MOVL C01070 V=800.0 PL=0
MOVL C01071 V=800.0 PL=0
MOVL C01072 V=800.0 PL=0
MOVL C01073 V=800.0 PL=0
MOVL C01074 V=800.0 PL=0
MOVL C01075 V=800.0 PL=0
MOVL C01076 V=800.0 PL=0
MOVL C01077 V=800.0 PL=0
MOVL C01078 V=800.0 PL=0
MOVL C01079 V=800.0 PL=0
MOVL C01080 V=800.0 PL=0
MOVL C01081 V=800.0 PL=0
MOVL C01082 V=800.0 PL=0
MOVL C01083 V=800.0 PL=0
MOVL C01084 V=800.0 PL=0
MOVL C01085 V=800.0 PL=0
MOVL C01086 V=800.0 PL=0
MOVL C01087 V=800.0 PL=0
MOVL C01088 V=800.0 PL=0
MOVL C01089 V=800.0 PL=0
MOVL C01090 V=800.0 PL=0
MOVL C01091 V=800.0 PL=0
MOVL C01092 V=800.0 PL=0
MOVL C01093 V=800.0 PL=0
MOVL C01094 V=800.0 PL=0
MOVL C01095 V=800.0 PL=0
MOVL C01096 V=800.0 PL=0
MOVL C01097 V=800.0 PL=0
MOVL C01098 V=800.0 PL=0
MOVL C01099 V=800.0 PL=0
MOVL C01100 V=800.0 PL=0
MOVL C01101 V=800.0 PL=0
MOVL C01102 V=800.0 PL=0
MOVL C01103 V=800.0 PL=0
MOVL C01104 V=800.0 PL=0
MOVL C01105 V=800.0 PL=0
MOVL C01106 V=800.0 PL=0
MOVL C01107 V=800.0 PL=0
MOVL C01108 V=800.0 PL=0
MOVL C01109 V=800.0 PL=0
MOVL C01110 V=800.0 PL=0
MOVL C01111 V=800.0 PL=0
MOVL C01112 V=800.0 PL=0
MOVL C01113 V=800.0 PL=0
MOVL C01114 V=800.0 PL=0
MOVL C01115 V=800.0 PL=0
MOVL C01116 V=800.0 PL=0
MOVL C01117 V=800.0 PL=0
MOVL C01118 V=800.0 PL=0
MOVL C01119 V=800.0 PL=0
MOVL C01120 V=800.0 PL=0
MOVL C01121 V=800.0 PL=0
MOVL C01122 V=800.0 PL=0
MOVL C01123 V=800.0 PL=0
MOVL C01124 V=800.0 PL=0
MOVL C01125 V=800.0 PL=0
MOVL C01126 V=800.0 PL=0
MOVL C01127 V=800.0 PL=0
MOVL C01128 V=800.0 PL=0
MOVL C01129 V=800.0 PL=0
MOVL C01130 V=800.0 PL=0
MOVL C01131 V=800.0 PL=0
MOVL C01132 V=800.0 PL=0
MOVL C01133 V=800.0 PL=0
MOVL C01134 V=800.0 PL=0
MOVL C01135 V=800.0 PL=0
MOVL C01136 V=800.0 PL=0
MOVL C01137 V=800.0 PL=0
MOVL C01138 V=800.0 PL=0
MOVL C01139 V=800.0 PL=0
MOVL C01140 V=800.0 PL=0
MOVL C01141 V=800.0 PL=0
MOVL C01142 V=800.0 PL=0
MOVL C01143 V=800.0 PL=0
MOVL C01144 V=800.0 PL=0
MOVL C01145 V=800.0 PL=0
MOVL C01146 V=800.0 PL=0
MOVL C01147 V=800.0 PL=0
MOVL C01148 V=800.0 PL=0
MOVL C01149 V=800.0 PL=0
MOVL C01150 V=800.0 PL=0
MOVL C01151 V=800.0 PL=0
MOVL C01152 V=800.0 PL=0
MOVL C01153 V=800.0 PL=0
MOVL C01154 V=800.0 PL=0
MOVL C01155 V=800.0 PL=0
MOVL C01156 V=800.0 PL=0
MOVL C01157 V=800.0 PL=0
MOVL C01158 V=800.0 PL=0
MOVL C01159 V=800.0 PL=0
MOVL C01160 V=800.0 PL=0
MOVL C01161 V=800.0 PL=0
MOVL C01162 V=800.0 PL=0
MOVL C01163 V=800.0 PL=0
MOVL C01164 V=800.0 PL=0
MOVL C01165 V=800.0 PL=0
MOVL C01166 V=800.0 PL=0
MOVL C01167 V=800.0 PL=0
MOVL C01168 V=800.0 PL=0
MOVL C01169 V=800.0 PL=0
MOVL C01170 V=800.0 PL=0
MOVL C01171 V=800.0 PL=0
MOVL C01172 V=800.0 PL=0
MOVL C01173 V=800.0 PL=0
MOVL C01174 V=800.0 PL=0
MOVL C01175 V=800.0 PL=0
MOVL C01176 V=800.0 PL=0
MOVL C01177 V=800.0 PL=0
MOVL C01178 V=800.0 PL=0
MOVL C01179 V=800.0 PL=0
MOVL C01180 V=800.0 PL=0
MOVL C01181 V=800.0 PL=0
MOVL C01182 V=800.0 PL=0
MOVL C01183 V=800.0 PL=0
MOVL C01184 V=800.0 PL=0
MOVL C01185 V=800.0 PL=0
MOVL C01186 V=800.0 PL=0
MOVL C01187 V=800.0 PL=0
MOVL C01188 V=800.0 PL=0
MOVL C01189 V=800.0 PL=0
MOVL C01190 V=800.0 PL=0
MOVL C01191 V=800.0 PL=0
MOVL C01192 V=800.0 PL=0
MOVL C01193 V=800.0 PL=0
MOVL C01194 V=800.0 PL=0
MOVL C01195 V=800.0 PL=0
MOVL C01196 V=800.0 PL=0
MOVL C01197 V=800.0 PL=0
MOVL C01198 V=800.0 PL=0
MOVL C01199 V=800.0 PL=0
MOVL C01200 V=800.0 PL=0
MOVL C01201 V=800.0 PL=0
MOVL C01202 V=800.0 PL=0
MOVL C01203 V=800.0 PL=0
MOVL C01204 V=800.0 PL=0
MOVL C01205 V=800.0 PL=0
MOVL C01206 V=800.0 PL=0
MOVL C01207 V=800.0 PL=0
MOVL C01208 V=800.0 PL=0
MOVL C01209 V=800.0 PL=0
MOVL C01210 V=800.0 PL=0
MOVL C01211 V=800.0 PL=0
MOVL C01212 V=800.0 PL=0
MOVL C01213 V=800.0 PL=0
MOVL C01214 V=800.0 PL=0
MOVL C01215 V=800.0 PL=0
MOVL C01216 V=800.0 PL=0
MOVL C01217 V=800.0 PL=0
MOVL C01218 V=800.0 PL=0
MOVL C01219 V=800.0 PL=0
MOVL C01220 V=800.0 PL=0
MOVL C01221 V=800.0 PL=0
MOVL C01222 V=800.0 PL=0
MOVL C01223 V=800.0 PL=0
MOVL C01224 V=800.0 PL=0
MOVL C01225 V=800.0 PL=0
MOVL C01226 V=800.0 PL=0
MOVL C01227 V=800.0 PL=0
MOVL C01228 V=800.0 PL=0
MOVL C01229 V=800.0 PL=0
MOVL C01230 V=800.0 PL=0
MOVL C01231 V=800.0 PL=0
MOVL C01232 V=800.0 PL=0
MOVL C01233 V=800.0 PL=0
MOVL C01234 V=800.0 PL=0
MOVL C01235 V=800.0 PL=0
MOVL C01236 V=800.0 PL=0
MOVL C01237 V=800.0 PL=0
MOVL C01238 V=800.0 PL=0
MOVL C01239 V=800.0 PL=0
MOVL C01240 V=800.0 PL=0
MOVL C01241 V=800.0 PL=0
MOVL C01242 V=800.0 PL=0
MOVL C01243 V=800.0 PL=0
MOVL C01244 V=800.0 PL=0
MOVL C01245 V=800.0 PL=0
MOVL C01246 V=800.0 PL=0
MOVL C01247 V=800.0 PL=0
MOVL C01248 V=800.0 PL=0
MOVL C01249 V=800.0 PL=0
MOVL C01250 V=800.0 PL=0
MOVL C01251 V=800.0 PL=0
MOVL C01252 V=800.0 PL=0
MOVL C01253 V=800.0 PL=0
MOVL C01254 V=800.0 PL=0
MOVL C01255 V=800.0 PL=0
MOVL C01256 V=800.0 PL=0
MOVL C01257 V=800.0 PL=0
MOVL C01258 V=800.0 PL=0
MOVL C01259 V=800.0 PL=0
MOVL C01260 V=800.0 PL=0
MOVL C01261 V=800.0 PL=0
MOVL C01262 V=800.0 PL=0
MOVL C01263 V=800.0 PL=0
MOVL C01264 V=800.0 PL=0
MOVL C01265 V=800.0 PL=0
MOVL C01266 V=800.0 PL=0
MOVL C01267 V=800.0 PL=0
MOVL C01268 V=800.0 PL=0
MOVL C01269 V=800.0 PL=0
MOVL C01270 V=800.0 PL=0
MOVL C01271 V=800.0 PL=0
MOVL C01272 V=800.0 PL=0
MOVL C01273 V=800.0 PL=0
MOVL C01274 V=800.0 PL=0
MOVL C01275 V=800.0 PL=0
MOVL C01276 V=800.0 PL=0
MOVL C01277 V=800.0 PL=0
MOVL C01278 V=800.0 PL=0
MOVL C01279 V=800.0 PL=0
MOVL C01280 V=800.0 PL=0
MOVL C01281 V=800.0 PL=0
MOVL C01282 V=800.0 PL=0
MOVL C01283 V=800.0 PL=0
MOVL C01284 V=800.0 PL=0
MOVL C01285 V=800.0 PL=0
MOVL C01286 V=800.0 PL=0
MOVL C01287 V=800.0 PL=0
MOVL C01288 V=800.0 PL=0
MOVL C01289 V=800.0 PL=0
MOVL C01290 V=800.0 PL=0
MOVL C01291 V=800.0 PL=0
MOVL C01292 V=800.0 PL=0
MOVL C01293 V=800.0 PL=0
MOVL C01294 V=800.0 PL=0
MOVL C01295 V=800.0 PL=0
MOVL C01296 V=800.0 PL=0
MOVL C01297 V=800.0 PL=0
MOVL C01298 V=800.0 PL=0
MOVL C01299 V=800.0 PL=0
MOVL C01300 V=800.0 PL=0
MOVL C01301 V=800.0 PL=0
MOVL C01302 V=800.0 PL=0
MOVL C01303 V=800.0 PL=0
MOVL C01304 V=800.0 PL=0
MOVL C01305 V=800.0 PL=0
MOVL C01306 V=800.0 PL=0
MOVL C01307 V=800.0 PL=0
MOVL C01308 V=800.0 PL=0
MOVL C01309 V=800.0 PL=0
MOVL C01310 V=800.0 PL=0
MOVL C01311 V=800.0 PL=0
MOVL C01312 V=800.0 PL=0
MOVL C01313 V=800.0 PL=0
MOVL C01314 V=800.0 PL=0
MOVL C01315 V=800.0 PL=0
MOVL C01316 V=800.0 PL=0
MOVL C01317 V=800.0 PL=0
MOVL C01318 V=800.0 PL=0
MOVL C01319 V=800.0 PL=0
MOVL C01320 V=800.0 PL=0
MOVL C01321 V=800.0 PL=0
MOVL C01322 V=800.0 PL=0
MOVL C01323 V=800.0 PL=0
MOVL C01324 V=800.0 PL=0
MOVL C01325 V=800.0 PL=0
MOVL C01326 V=800.0 PL=0
MOVL C01327 V=800.0 PL=0
MOVL C01328 V=800.0 PL=0
MOVL C01329 V=800.0 PL=0
MOVL C01330 V=800.0 PL=0
MOVL C01331 V=800.0 PL=0
MOVL C01332 V=800.0 PL=0
MOVL C01333 V=800.0 PL=0
MOVL C01334 V=800.0 PL=0
MOVL C01335 V=800.0 PL=0
MOVL C01336 V=800.0 PL=0
MOVL C01337 V=800.0 PL=0
MOVL C01338 V=800.0 PL=0
MOVL C01339 V=800.0 PL=0
MOVL C01340 V=800.0 PL=0
MOVL C01341 V=800.0 PL=0
MOVL C01342 V=800.0 PL=0
MOVL C01343 V=800.0 PL=0
MOVL C01344 V=800.0 PL=0
MOVL C01345 V=800.0 PL=0
MOVL C01346 V=800.0 PL=0
MOVL C01347 V=800.0 PL=0
MOVL C01348 V=800.0 PL=0
MOVL C01349 V=800.0 PL=0
MOVL C01350 V=800.0 PL=0
MOVL C01351 V=800.0 PL=0
MOVL C01352 V=800.0 PL=0
MOVL C01353 V=800.0 PL=0
MOVL C01354 V=800.0 PL=0
MOVL C01355 V=800.0 PL=0
MOVL C01356 V=800.0 PL=0
MOVL C01357 V=800.0 PL=0
MOVL C01358 V=800.0 PL=0
MOVL C01359 V=800.0 PL=0
MOVL C01360 V=800.0 PL=0
MOVL C01361 V=800.0 PL=0
MOVL C01362 V=800.0 PL=0
MOVL C01363 V=800.0 PL=0
MOVL C01364 V=800.0 PL=0
MOVL C01365 V=800.0 PL=0
MOVL C01366 V=800.0 PL=0
MOVL C01367 V=800.0 PL=0
MOVL C01368 V=800.0 PL=0
MOVL C01369 V=800.0 PL=0
MOVL C01370 V=800.0 PL=0
MOVL C01371 V=800.0 PL=0
MOVL C01372 V=800.0 PL=0
MOVL C01373 V=800.0 PL=0
MOVL C01374 V=800.0 PL=0
MOVL C01375 V=800.0 PL=0
MOVL C01376 V=800.0 PL=0
MOVL C01377 V=800.0 PL=0
MOVL C01378 V=800.0 PL=0
MOVL C01379 V=800.0 PL=0
MOVL C01380 V=800.0 PL=0
MOVL C01381 V=800.0 PL=0
MOVL C01382 V=800.0 PL=0
MOVL C01383 V=800.0 PL=0
MOVL C01384 V=800.0 PL=0
MOVL C01385 V=800.0 PL=0
MOVL C01386 V=800.0 PL=0
MOVL C01387 V=800.0 PL=0
MOVL C01388 V=800.0 PL=0
MOVL C01389 V=800.0 PL=0
MOVL C01390 V=800.0 PL=0
MOVL C01391 V=800.0 PL=0
MOVL C01392 V=800.0 PL=0
MOVL C01393 V=800.0 PL=0
MOVL C01394 V=800.0 PL=0
MOVL C01395 V=800.0 PL=0
MOVL C01396 V=800.0 PL=0
MOVL C01397 V=800.0 PL=0
MOVL C01398 V=800.0 PL=0
MOVL C01399 V=800.0 PL=0
MOVL C01400 V=800.0 PL=0
MOVL C01401 V=800.0 PL=0
MOVL C01402 V=800.0 PL=0
MOVL C01403 V=800.0 PL=0
MOVL C01404 V=800.0 PL=0
MOVL C01405 V=800.0 PL=0
MOVL C01406 V=800.0 PL=0
MOVL C01407 V=800.0 PL=0
MOVL C01408 V=800.0 PL=0
MOVL C01409 V=800.0 PL=0
MOVL C01410 V=800.0 PL=0
MOVL C01411 V=800.0 PL=0
MOVL C01412 V=800.0 PL=0
MOVL C01413 V=800.0 PL=0
MOVL C01414 V=800.0 PL=0
MOVL C01415 V=800.0 PL=0
MOVL C01416 V=800.0 PL=0
MOVL C01417 V=800.0 PL=0
MOVL C01418 V=800.0 PL=0
MOVL C01419 V=800.0 PL=0
MOVL C01420 V=800.0 PL=0
MOVL C01421 V=800.0 PL=0
MOVL C01422 V=800.0 PL=0
MOVL C01423 V=800.0 PL=0
MOVL C01424 V=800.0 PL=0
MOVL C01425 V=800.0 PL=0
MOVL C01426 V=800.0 PL=0
MOVL C01427 V=800.0 PL=0
MOVL C01428 V=800.0 PL=0
MOVL C01429 V=800.0 PL=0
MOVL C01430 V=800.0 PL=0
MOVL C01431 V=800.0 PL=0
MOVL C01432 V=800.0 PL=0
MOVL C01433 V=800.0 PL=0
MOVL C01434 V=800.0 PL=0
MOVL C01435 V=800.0 PL=0
MOVL C01436 V=800.0 PL=0
MOVL C01437 V=800.0 PL=0
MOVL C01438 V=800.0 PL=0
MOVL C01439 V=800.0 PL=0
MOVL C01440 V=800.0 PL=0
MOVL C01441 V=800.0 PL=0
MOVL C01442 V=800.0 PL=0
MOVL C01443 V=800.0 PL=0
MOVL C01444 V=800.0 PL=0
MOVL C01445 V=800.0 PL=0
MOVL C01446 V=800.0 PL=0
MOVL C01447 V=800.0 PL=0
MOVL C01448 V=800.0 PL=0
MOVL C01449 V=800.0 PL=0
MOVL C01450 V=800.0 PL=0
MOVL C01451 V=800.0 PL=0
MOVL C01452 V=800.0 PL=0
MOVL C01453 V=800.0 PL=0
MOVL C01454 V=800.0 PL=0
MOVL C01455 V=800.0 PL=0
MOVL C01456 V=800.0 PL=0
MOVL C01457 V=800.0 PL=0
MOVL C01458 V=800.0 PL=0
MOVL C01459 V=800.0 PL=0
MOVL C01460 V=800.0 PL=0
MOVL C01461 V=800.0 PL=0
MOVL C01462 V=800.0 PL=0
MOVL C01463 V=800.0 PL=0
MOVL C01464 V=800.0 PL=0
MOVL C01465 V=800.0 PL=0
MOVL C01466 V=800.0 PL=0
MOVL C01467 V=800.0 PL=0
MOVL C01468 V=800.0 PL=0
MOVL C01469 V=800.0 PL=0
MOVL C01470 V=800.0 PL=0
MOVL C01471 V=800.0 PL=0
MOVL C01472 V=800.0 PL=0
MOVL C01473 V=800.0 PL=0
MOVL C01474 V=800.0 PL=0
MOVL C01475 V=800.0 PL=0
MOVL C01476 V=800.0 PL=0
MOVL C01477 V=800.0 PL=0
MOVL C01478 V=800.0 PL=0
MOVL C01479 V=800.0 PL=0
MOVL C01480 V=800.0 PL=0
MOVL C01481 V=800.0 PL=0
MOVL C01482 V=800.0 PL=0
MOVL C01483 V=800.0 PL=0
MOVL C01484 V=800.0 PL=0
MOVL C01485 V=800.0 PL=0
MOVL C01486 V=800.0 PL=0
MOVL C01487 V=800.0 PL=0
MOVL C01488 V=800.0 PL=0
MOVL C01489 V=800.0 PL=0
MOVL C01490 V=800.0 PL=0
MOVL C01491 V=800.0 PL=0
MOVL C01492 V=800.0 PL=0
MOVL C01493 V=800.0 PL=0
MOVL C01494 V=800.0 PL=0
MOVL C01495 V=800.0 PL=0
MOVL C01496 V=800.0 PL=0
MOVL C01497 V=800.0 PL=0
MOVL C01498 V=800.0 PL=0
MOVL C01499 V=800.0 PL=0
MOVL C01500 V=800.0 PL=0
MOVL C01501 V=800.0 PL=0
MOVL C01502 V=800.0 PL=0
MOVL C01503 V=800.0 PL=0
MOVL C01504 V=800.0 PL=0
MOVL C01505 V=800.0 PL=0
MOVL C01506 V=800.0 PL=0
MOVL C01507 V=800.0 PL=0
MOVL C01508 V=800.0 PL=0
MOVL C01509 V=800.0 PL=0
MOVL C01510 V=800.0 PL=0
MOVL C01511 V=800.0 PL=0
MOVL C01512 V=800.0 PL=0
MOVL C01513 V=800.0 PL=0
MOVL C01514 V=800.0 PL=0
MOVL C01515 V=800.0 PL=0
MOVL C01516 V=800.0 PL=0
MOVL C01517 V=800.0 PL=0
MOVL C01518 V=800.0 PL=0
MOVL C01519 V=800.0 PL=0
MOVL C01520 V=800.0 PL=0
MOVL C01521 V=800.0 PL=0
MOVL C01522 V=800.0 PL=0
MOVL C01523 V=800.0 PL=0
MOVL C01524 V=800.0 PL=0
MOVL C01525 V=800.0 PL=0
MOVL C01526 V=800.0 PL=0
MOVL C01527 V=800.0 PL=0
MOVL C01528 V=800.0 PL=0
MOVL C01529 V=800.0 PL=0
MOVL C01530 V=800.0 PL=0
MOVL C01531 V=800.0 PL=0
MOVL C01532 V=800.0 PL=0
MOVL C01533 V=800.0 PL=0
MOVL C01534 V=800.0 PL=0
MOVL C01535 V=800.0 PL=0
MOVL C01536 V=800.0 PL=0
MOVL C01537 V=800.0 PL=0
MOVL C01538 V=800.0 PL=0
MOVL C01539 V=800.0 PL=0
MOVL C01540 V=800.0 PL=0
MOVL C01541 V=800.0 PL=0
MOVL C01542 V=800.0 PL=0
MOVL C01543 V=800.0 PL=0
MOVL C01544 V=800.0 PL=0
MOVL C01545 V=800.0 PL=0
MOVL C01546 V=800.0 PL=0
MOVL C01547 V=800.0 PL=0
MOVL C01548 V=800.0 PL=0
MOVL C01549 V=800.0 PL=0
MOVL C01550 V=800.0 PL=0
MOVL C01551 V=800.0 PL=0
MOVL C01552 V=800.0 PL=0
MOVL C01553 V=800.0 PL=0
MOVL C01554 V=800.0 PL=0
MOVL C01555 V=800.0 PL=0
MOVL C01556 V=800.0 PL=0
MOVL C01557 V=800.0 PL=0
MOVL C01558 V=800.0 PL=0
MOVL C01559 V=800.0 PL=0
MOVL C01560 V=800.0 PL=0
MOVL C01561 V=800.0 PL=0
MOVL C01562 V=800.0 PL=0
MOVL C01563 V=800.0 PL=0
MOVL C01564 V=800.0 PL=0
MOVL C01565 V=800.0 PL=0
MOVL C01566 V=800.0 PL=0
MOVL C01567 V=800.0 PL=0
MOVL C01568 V=800.0 PL=0
MOVL C01569 V=800.0 PL=0
MOVL C01570 V=800.0 PL=0
MOVL C01571 V=800.0 PL=0
MOVL C01572 V=800.0 PL=0
MOVL C01573 V=800.0 PL=0
MOVL C01574 V=800.0 PL=0
MOVL C01575 V=800.0 PL=0
MOVL C01576 V=800.0 PL=0
MOVL C01577 V=800.0 PL=0
MOVL C01578 V=800.0 PL=0
MOVL C01579 V=800.0 PL=0
MOVL C01580 V=800.0 PL=0
MOVL C01581 V=800.0 PL=0
MOVL C01582 V=800.0 PL=0
MOVL C01583 V=800.0 PL=0
MOVL C01584 V=800.0 PL=0
MOVL C01585 V=800.0 PL=0
MOVL C01586 V=800.0 PL=0
MOVL C01587 V=800.0 PL=0
MOVL C01588 V=800.0 PL=0
MOVL C01589 V=800.0 PL=0
MOVL C01590 V=800.0 PL=0
MOVL C01591 V=800.0 PL=0
MOVL C01592 V=800.0 PL=0
MOVL C01593 V=800.0 PL=0
MOVL C01594 V=800.0 PL=0
MOVL C01595 V=800.0 PL=0
MOVL C01596 V=800.0 PL=0
MOVL C01597 V=800.0 PL=0
MOVL C01598 V=800.0 PL=0
MOVL C01599 V=800.0 PL=0
MOVL C01600 V=800.0 PL=0
MOVL C01601 V=800.0 PL=0
MOVL C01602 V=800.0 PL=0
MOVL C01603 V=800.0 PL=0
MOVL C01604 V=800.0 PL=0
MOVL C01605 V=800.0 PL=0
MOVL C01606 V=800.0 PL=0
MOVL C01607 V=800.0 PL=0
MOVL C01608 V=800.0 PL=0
MOVL C01609 V=800.0 PL=0
MOVL C01610 V=800.0 PL=0
MOVL C01611 V=800.0 PL=0
MOVL C01612 V=800.0 PL=0
MOVL C01613 V=800.0 PL=0
MOVL C01614 V=800.0 PL=0
MOVL C01615 V=800.0 PL=0
MOVL C01616 V=800.0 PL=0
MOVL C01617 V=800.0 PL=0
MOVL C01618 V=800.0 PL=0
MOVL C01619 V=800.0 PL=0
MOVL C01620 V=800.0 PL=0
MOVL C01621 V=800.0 PL=0
MOVL C01622 V=800.0 PL=0
MOVL C01623 V=800.0 PL=0
MOVL C01624 V=800.0 PL=0
MOVL C01625 V=800.0 PL=0
MOVL C01626 V=800.0 PL=0
MOVL C01627 V=800.0 PL=0
MOVL C01628 V=800.0 PL=0
MOVL C01629 V=800.0 PL=0
MOVL C01630 V=800.0 PL=0
MOVL C01631 V=800.0 PL=0
MOVL C01632 V=800.0 PL=0
MOVL C01633 V=800.0 PL=0
MOVL C01634 V=800.0 PL=0
MOVL C01635 V=800.0 PL=0
MOVL C01636 V=800.0 PL=0
MOVL C01637 V=800.0 PL=0
MOVL C01638 V=800.0 PL=0
MOVL C01639 V=800.0 PL=0
MOVL C01640 V=800.0 PL=0
MOVL C01641 V=800.0 PL=0
MOVL C01642 V=800.0 PL=0
MOVL C01643 V=800.0 PL=0
MOVL C01644 V=800.0 PL=0
MOVL C01645 V=800.0 PL=0
MOVL C01646 V=800.0 PL=0
MOVL C01647 V=800.0 PL=0
MOVL C01648 V=800.0 PL=0
MOVL C01649 V=800.0 PL=0
MOVL C01650 V=800.0 PL=0
MOVL C01651 V=800.0 PL=0
MOVL C01652 V=800.0 PL=0
MOVL C01653 V=800.0 PL=0
MOVL C01654 V=800.0 PL=0
MOVL C01655 V=800.0 PL=0
MOVL C01656 V=800.0 PL=0
MOVL C01657 V=800.0 PL=0
MOVL C01658 V=800.0 PL=0
MOVL C01659 V=800.0 PL=0
MOVL C01660 V=800.0 PL=0
MOVL C01661 V=800.0 PL=0
MOVL C01662 V=800.0 PL=0
MOVL C01663 V=800.0 PL=0
MOVL C01664 V=800.0 PL=0
MOVL C01665 V=800.0 PL=0
MOVL C01666 V=800.0 PL=0
MOVL C01667 V=800.0 PL=0
MOVL C01668 V=800.0 PL=0
MOVL C01669 V=800.0 PL=0
MOVL C01670 V=800.0 PL=0
MOVL C01671 V=800.0 PL=0
MOVL C01672 V=800.0 PL=0
MOVL C01673 V=800.0 PL=0
MOVL C01674 V=800.0 PL=0
MOVL C01675 V=800.0 PL=0
MOVL C01676 V=800.0 PL=0
MOVL C01677 V=800.0 PL=0
MOVL C01678 V=800.0 PL=0
MOVL C01679 V=800.0 PL=0
MOVL C01680 V=800.0 PL=0
MOVL C01681 V=800.0 PL=0
MOVL C01682 V=800.0 PL=0
MOVL C01683 V=800.0 PL=0
MOVL C01684 V=800.0 PL=0
MOVL C01685 V=800.0 PL=0
MOVL C01686 V=800.0 PL=0
MOVL C01687 V=800.0 PL=0
MOVL C01688 V=800.0 PL=0
MOVL C01689 V=800.0 PL=0
MOVL C01690 V=800.0 PL=0
MOVL C01691 V=800.0 PL=0
MOVL C01692 V=800.0 PL=0
MOVL C01693 V=800.0 PL=0
MOVL C01694 V=800.0 PL=0
MOVL C01695 V=800.0 PL=0
MOVL C01696 V=800.0 PL=0
MOVL C01697 V=800.0 PL=0
MOVL C01698 V=800.0 PL=0
MOVL C01699 V=800.0 PL=0
MOVL C01700 V=800.0 PL=0
MOVL C01701 V=800.0 PL=0
MOVL C01702 V=800.0 PL=0
MOVL C01703 V=800.0 PL=0
MOVL C01704 V=800.0 PL=0
MOVL C01705 V=800.0 PL=0
MOVL C01706 V=800.0 PL=0
MOVL C01707 V=800.0 PL=0
MOVL C01708 V=800.0 PL=0
MOVL C01709 V=800.0 PL=0
MOVL C01710 V=800.0 PL=0
MOVL C01711 V=800.0 PL=0
MOVL C01712 V=800.0 PL=0
MOVL C01713 V=800.0 PL=0
MOVL C01714 V=800.0 PL=0
MOVL C01715 V=800.0 PL=0
MOVL C01716 V=800.0 PL=0
MOVL C01717 V=800.0 PL=0
MOVL C01718 V=800.0 PL=0
MOVL C01719 V=800.0 PL=0
MOVL C01720 V=800.0 PL=0
MOVL C01721 V=800.0 PL=0
MOVL C01722 V=800.0 PL=0
MOVL C01723 V=800.0 PL=0
MOVL C01724 V=800.0 PL=0
MOVL C01725 V=800.0 PL=0
MOVL C01726 V=800.0 PL=0
MOVL C01727 V=800.0 PL=0
MOVL C01728 V=800.0 PL=0
MOVL C01729 V=800.0 PL=0
MOVL C01730 V=800.0 PL=0
MOVL C01731 V=800.0 PL=0
MOVL C01732 V=800.0 PL=0
MOVL C01733 V=800.0 PL=0
MOVL C01734 V=800.0 PL=0
MOVL C01735 V=800.0 PL=0
MOVL C01736 V=800.0 PL=0
MOVL C01737 V=800.0 PL=0
MOVL C01738 V=800.0 PL=0
MOVL C01739 V=800.0 PL=0
MOVL C01740 V=800.0 PL=0
MOVL C01741 V=800.0 PL=0
MOVL C01742 V=800.0 PL=0
MOVL C01743 V=800.0 PL=0
MOVL C01744 V=800.0 PL=0
MOVL C01745 V=800.0 PL=0
MOVL C01746 V=800.0 PL=0
MOVL C01747 V=800.0 PL=0
MOVL C01748 V=800.0 PL=0
MOVL C01749 V=800.0 PL=0
MOVL C01750 V=800.0 PL=0
MOVL C01751 V=800.0 PL=0
MOVL C01752 V=800.0 PL=0
MOVL C01753 V=800.0 PL=0
MOVL C01754 V=800.0 PL=0
MOVL C01755 V=800.0 PL=0
MOVL C01756 V=800.0 PL=0
MOVL C01757 V=800.0 PL=0
MOVL C01758 V=800.0 PL=0
MOVL C01759 V=800.0 PL=0
MOVL C01760 V=800.0 PL=0
MOVL C01761 V=800.0 PL=0
MOVL C01762 V=800.0 PL=0
MOVL C01763 V=800.0 PL=0
MOVL C01764 V=800.0 PL=0
MOVL C01765 V=800.0 PL=0
MOVL C01766 V=800.0 PL=0
MOVL C01767 V=800.0 PL=0
MOVL C01768 V=800.0 PL=0
MOVL C01769 V=800.0 PL=0
MOVL C01770 V=800.0 PL=0
MOVL C01771 V=800.0 PL=0
MOVL C01772 V=800.0 PL=0
MOVL C01773 V=800.0 PL=0
MOVL C01774 V=800.0 PL=0
MOVL C01775 V=800.0 PL=0
MOVL C01776 V=800.0 PL=0
MOVL C01777 V=800.0 PL=0
MOVL C01778 V=800.0 PL=0
MOVL C01779 V=800.0 PL=0
MOVL C01780 V=800.0 PL=0
MOVL C01781 V=800.0 PL=0
MOVL C01782 V=800.0 PL=0
MOVL C01783 V=800.0 PL=0
MOVL C01784 V=800.0 PL=0
MOVL C01785 V=800.0 PL=0
MOVL C01786 V=800.0 PL=0
MOVL C01787 V=800.0 PL=0
MOVL C01788 V=800.0 PL=0
MOVL C01789 V=800.0 PL=0
MOVL C01790 V=800.0 PL=0
MOVL C01791 V=800.0 PL=0
MOVL C01792 V=800.0 PL=0
MOVL C01793 V=800.0 PL=0
MOVL C01794 V=800.0 PL=0
MOVL C01795 V=800.0 PL=0
MOVL C01796 V=800.0 PL=0
MOVL C01797 V=800.0 PL=0
MOVL C01798 V=800.0 PL=0
MOVL C01799 V=800.0 PL=0
MOVL C01800 V=800.0 PL=0
MOVL C01801 V=800.0 PL=0
MOVL C01802 V=800.0 PL=0
MOVL C01803 V=800.0 PL=0
MOVL C01804 V=800.0 PL=0
MOVL C01805 V=800.0 PL=0
MOVL C01806 V=800.0 PL=0
MOVL C01807 V=800.0 PL=0
MOVL C01808 V=800.0 PL=0
MOVL C01809 V=800.0 PL=0
MOVL C01810 V=800.0 PL=0
MOVL C01811 V=800.0 PL=0
MOVL C01812 V=800.0 PL=0
MOVL C01813 V=800.0 PL=0
MOVL C01814 V=800.0 PL=0
MOVL C01815 V=800.0 PL=0
MOVL C01816 V=800.0 PL=0
MOVL C01817 V=800.0 PL=0
MOVL C01818 V=800.0 PL=0
MOVL C01819 V=800.0 PL=0
MOVL C01820 V=800.0 PL=0
MOVL C01821 V=800.0 PL=0
MOVL C01822 V=800.0 PL=0
MOVL C01823 V=800.0 PL=0
MOVL C01824 V=800.0 PL=0
MOVL C01825 V=800.0 PL=0
MOVL C01826 V=800.0 PL=0
MOVL C01827 V=800.0 PL=0
MOVL C01828 V=800.0 PL=0
MOVL C01829 V=800.0 PL=0
MOVL C01830 V=800.0 PL=0
MOVL C01831 V=800.0 PL=0
MOVL C01832 V=800.0 PL=0
MOVL C01833 V=800.0 PL=0
MOVL C01834 V=800.0 PL=0
MOVL C01835 V=800.0 PL=0
MOVL C01836 V=800.0 PL=0
MOVL C01837 V=800.0 PL=0
MOVL C01838 V=800.0 PL=0
MOVL C01839 V=800.0 PL=0
MOVL C01840 V=800.0 PL=0
MOVL C01841 V=800.0 PL=0
MOVL C01842 V=800.0 PL=0
MOVL C01843 V=800.0 PL=0
MOVL C01844 V=800.0 PL=0
MOVL C01845 V=800.0 PL=0
MOVL C01846 V=800.0 PL=0
MOVL C01847 V=800.0 PL=0
MOVL C01848 V=800.0 PL=0
MOVL C01849 V=800.0 PL=0
MOVL C01850 V=800.0 PL=0
MOVL C01851 V=800.0 PL=0
MOVL C01852 V=800.0 PL=0
MOVL C01853 V=800.0 PL=0
MOVL C01854 V=800.0 PL=0
MOVL C01855 V=800.0 PL=0
MOVL C01856 V=800.0 PL=0
MOVL C01857 V=800.0 PL=0
MOVL C01858 V=800.0 PL=0
MOVL C01859 V=800.0 PL=0
MOVL C01860 V=800.0 PL=0
MOVL C01861 V=800.0 PL=0
MOVL C01862 V=800.0 PL=0
MOVL C01863 V=800.0 PL=0
MOVL C01864 V=800.0 PL=0
MOVL C01865 V=800.0 PL=0
MOVL C01866 V=800.0 PL=0
MOVL C01867 V=800.0 PL=0
MOVL C01868 V=800.0 PL=0
MOVL C01869 V=800.0 PL=0
MOVL C01870 V=800.0 PL=0
MOVL C01871 V=800.0 PL=0
MOVL C01872 V=800.0 PL=0
MOVL C01873 V=800.0 PL=0
MOVL C01874 V=800.0 PL=0
MOVL C01875 V=800.0 PL=0
MOVL C01876 V=800.0 PL=0
MOVL C01877 V=800.0 PL=0
MOVL C01878 V=800.0 PL=0
MOVL C01879 V=800.0 PL=0
MOVL C01880 V=800.0 PL=0
MOVL C01881 V=800.0 PL=0
MOVL C01882 V=800.0 PL=0
